RoboDK station: kr30 cnc 071219 julian curve.rdk

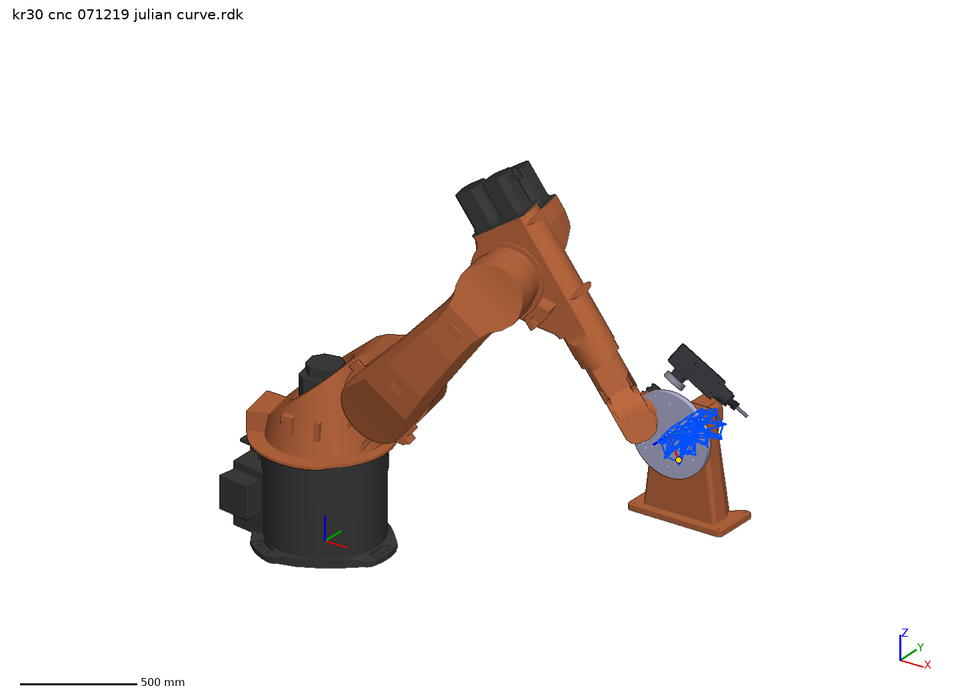
[picture v0: the station drawn from its stored meshes, robots at their saved joint values, targets as dots, program paths as lines]
Station kr30 cnc 071219 julian curve. Poses are relative to the parent item; angles as X-Y-Z fixed-axis rotations.
  - machining project Curve settings: C:/Temp/temp3/RhinoProject.stl | rotZ(0) | rotX(0)*rotY(0) | rotz(0) | onStart | onPathStart | onApproach | onPoint | onRetract | onFinish | onPathFinish | M_RunCode(%1)
  - frame KUKA KP1 MD250 Base at (0, 0, 0) mm
    - robot GIGASHEEN TURNTABLE OF DEATH: 1 axes, payload 250 kg
        modified DH rows (alpha deg, a mm, theta deg, d mm): 0, 0, 0, 0
        base shift (1587.22, 296.05, 828) mm, rotated rx 0 ry 90 rz -90 deg
        joint limits [-3600] to [3600]; home [0]; saved at [-332.14]
      - frame Reference Rhino at (0, 0, 0) mm
        - object RhinoPart at (0, -260, 100) mm
        - object Test Piece at (0, 0, 0) mm, geometry from Test Piece.stp
  - frame KUKA KR 30 HA Base at (0, 0, 0) mm
    - robot KUKA KR 30 HA: 6 axes, payload 30 kg, reach 2033 mm, repeatability 0.05 mm, weight 665 kg
        modified DH rows (alpha deg, a mm, theta deg, d mm): 0, 0, 0, 815; -90, 350, 0, 0; 0, 850, -90, 0; -90, 145, 0, 820; 90, 0, 0, 0; -90, 0, 180, 170
        joint limits [-185, -135, -120, -350, -119, -350] to [185, 35, 158, 350, 119, 350]; home [0, -90, 90, 0, 0, 0]; saved at [-11.373, -50.021, 107.833, -147.844, 108.332, -176.467]
      - tool 1/2" End Mill TCP, TCP at (337.71, -2.2, 160.57) mm, rotated rx 0 ry 90 rz 0 deg, size 415.8 x 102 x 153.6 mm
  - machining project RhinoPart Settings: rotZ(0) | rotX(90)*rotY(-155) | rotz(0)
  - program RhinoPart (1768 instructions, listed below)
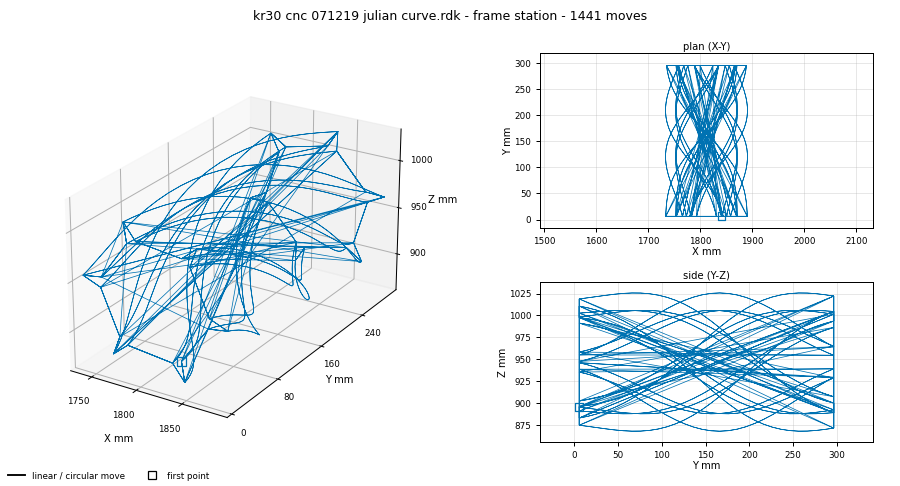
[picture p0: tool path of kr30 cnc 071219 julian curve.rdk in frame station, 1441 of 1441 moves have a stored position in this frame; points joined in program order, loops and branches not executed]

--- program RhinoPart (robot KUKA KR 30 HA) ---
  Set Ref.: Reference Rhino
  Set Tool: 1/2" End Mill TCP
  Show 1/2" End Mill TCP
  Set speed (1000.0 mm/s)
  MoveJ 1 to (58.93, 255.88, 290) mm, rotated rx -90 ry -25 rz 136 deg; joints [-2.265, -48.411, 103.049, -142.26, 108.636, -182.753, -175.998]
  MoveL 2 to (58.93, 255.88, 290) mm, rotated rx -90 ry -25 rz 136 deg; joints [-2.265, -48.411, 103.049, -142.26, 108.636, -182.753, -175.998]
  MoveL 3 to (58.93, 255.88, 290) mm, rotated rx -90 ry -25 rz 136 deg; joints [-2.265, -48.411, 103.049, -142.26, 108.636, -182.753, -175.998]
  Set speed (60.0 mm/s)
  MoveL 4 to (37.11, 300.24, 290) mm, rotated rx -90 ry -25 rz -172.69 deg; joints [-2.265, -48.205, 103.066, -142.213, 108.813, -182.608, -227.315]
  Set speed (1000.0 mm/s)
  MoveL 5 to (37.11, 300.24, 290) mm, rotated rx -90 ry -25 rz -172.69 deg; joints [-2.265, -48.205, 103.066, -142.213, 108.813, -182.608, -227.315]
  Set speed (1000.0 mm/s)
  MoveL 6 to (-37.11, 208.63, 290) mm, rotated rx -90 ry -25 rz 14.16 deg; joints [-2.265, -48.614, 103.03, -142.305, 108.461, -182.896, -54.156]
  MoveL 7 to (-37.11, 208.63, 290) mm, rotated rx -90 ry -25 rz 14.16 deg; joints [-2.265, -48.614, 103.03, -142.305, 108.461, -182.896, -54.156]
  Set speed (60.0 mm/s)
  MoveL 8 to (-58.93, 252.99, 290) mm, rotated rx -90 ry -25 rz -33.22 deg; joints [-2.265, -48.424, 103.048, -142.262, 108.625, -182.762, -6.784]
  Set speed (1000.0 mm/s)
  MoveL 9 to (-58.93, 252.99, 290) mm, rotated rx -90 ry -25 rz -33.22 deg; joints [-2.265, -48.424, 103.048, -142.262, 108.625, -182.762, -6.784]
  Set speed (1000.0 mm/s)
  MoveL 10 to (21.11, 199.39, 290) mm, rotated rx -90 ry -25 rz 69.21 deg; joints [-2.265, -48.652, 103.027, -142.314, 108.428, -182.923, -109.206]
  MoveL 11 to (21.11, 199.39, 290) mm, rotated rx -90 ry -25 rz 69.21 deg; joints [-2.265, -48.652, 103.027, -142.314, 108.428, -182.923, -109.206]
  Set speed (60.0 mm/s)
  MoveL 12 to (34.79, 183.72, 290) mm, rotated rx -90 ry -25 rz 74.51 deg; joints [-2.265, -49.571, 102.922, -142.517, 107.617, -183.579, -114.515]
  Set speed (1000.0 mm/s)
  MoveL 13 to (34.79, 183.72, 290) mm, rotated rx -90 ry -25 rz 74.51 deg; joints [-2.265, -49.571, 102.922, -142.517, 107.617, -183.579, -114.515]
  Set speed (1000.0 mm/s)
  MoveL 14 to (21.11, 199.39, 290) mm, rotated rx -90 ry -25 rz 69.21 deg; joints [-2.265, -48.652, 103.027, -142.314, 108.428, -182.923, -109.206]
  MoveL 15 to (21.11, 199.39, 290) mm, rotated rx -90 ry -25 rz 69.21 deg; joints [-2.265, -48.652, 103.027, -142.314, 108.428, -182.923, -109.206]
  Set speed (60.0 mm/s)
  MoveL 16 to (-28.22, 202.67, 290) mm, rotated rx -90 ry -25 rz 23.79 deg; joints [-2.265, -48.639, 103.028, -142.311, 108.44, -182.913, -63.793]
  Set speed (1000.0 mm/s)
  MoveL 17 to (-28.22, 202.67, 290) mm, rotated rx -90 ry -25 rz 23.79 deg; joints [-2.265, -48.639, 103.028, -142.311, 108.44, -182.913, -63.793]
  Set speed (1000.0 mm/s)
  MoveL 18 to (-43.85, 188.95, 290) mm, rotated rx -90 ry -25 rz 18.32 deg; joints [-2.265, -49.555, 102.924, -142.513, 107.631, -183.568, -58.321]
  MoveL 19 to (-43.85, 188.95, 290) mm, rotated rx -90 ry -25 rz 18.32 deg; joints [-2.265, -49.555, 102.924, -142.513, 107.631, -183.568, -58.321]
  Set speed (60.0 mm/s)
  MoveL 20 to (-28.22, 202.67, 290) mm, rotated rx -90 ry -25 rz 23.79 deg; joints [-2.265, -48.639, 103.028, -142.311, 108.44, -182.913, -63.793]
  Set speed (1000.0 mm/s)
  MoveL 21 to (-28.22, 202.67, 290) mm, rotated rx -90 ry -25 rz 23.79 deg; joints [-2.265, -48.639, 103.028, -142.311, 108.44, -182.913, -63.793]
  Set speed (1000.0 mm/s)
  MoveL 22 to (-43.85, 188.95, 290) mm, rotated rx -90 ry -25 rz 18.32 deg; joints [-2.265, -49.555, 102.924, -142.513, 107.631, -183.568, -58.321]
  MoveL 23 to (-43.85, 188.95, 290) mm, rotated rx -90 ry -25 rz 18.32 deg; joints [-2.265, -49.555, 102.924, -142.513, 107.631, -183.568, -58.321]
  Set speed (60.0 mm/s)
  MoveL 24 to (-37.11, 208.63, 290) mm, rotated rx -90 ry -25 rz 14.16 deg; joints [-2.265, -48.614, 103.03, -142.305, 108.461, -182.896, -54.156]
  Set speed (1000.0 mm/s)
  MoveL 25 to (-37.11, 208.63, 290) mm, rotated rx -90 ry -25 rz 14.16 deg; joints [-2.265, -48.614, 103.03, -142.305, 108.461, -182.896, -54.156]
  Set speed (1000.0 mm/s)
  MoveL 26 to (-78.63, 259.66, 290) mm, rotated rx -90 ry -25 rz -39.75 deg; joints [-2.265, -49.329, 102.952, -142.464, 107.833, -183.405, -0.245]
  MoveL 27 to (-78.63, 259.66, 290) mm, rotated rx -90 ry -25 rz -39.75 deg; joints [-2.265, -49.329, 102.952, -142.464, 107.833, -183.405, -0.245]
  Set speed (60.0 mm/s)
  MoveL 28 to (-58.93, 252.99, 290) mm, rotated rx -90 ry -25 rz -33.22 deg; joints [-2.265, -48.424, 103.048, -142.262, 108.625, -182.762, -6.784]
  Set speed (1000.0 mm/s)
  MoveL 29 to (-58.93, 252.99, 290) mm, rotated rx -90 ry -25 rz -33.22 deg; joints [-2.265, -48.424, 103.048, -142.262, 108.625, -182.762, -6.784]
  Set speed (1000.0 mm/s)
  MoveL 30 to (-78.63, 259.66, 290) mm, rotated rx -90 ry -25 rz -39.75 deg; joints [-2.265, -49.329, 102.952, -142.464, 107.833, -183.405, -0.245]
  MoveL 31 to (-78.63, 259.66, 290) mm, rotated rx -90 ry -25 rz -39.75 deg; joints [-2.265, -49.329, 102.952, -142.464, 107.833, -183.405, -0.245]
  Set speed (60.0 mm/s)
  MoveL 32 to (-58.22, 263.67, 290) mm, rotated rx -90 ry -25 rz -43.61 deg; joints [-2.265, -48.376, 103.052, -142.252, 108.666, -182.728, 3.606]
  Set speed (1000.0 mm/s)
  MoveL 33 to (-58.22, 263.67, 290) mm, rotated rx -90 ry -25 rz -43.61 deg; joints [-2.265, -48.376, 103.052, -142.252, 108.666, -182.728, 3.606]
  Set speed (1000.0 mm/s)
  MoveL 34 to (-30.72, 304.75, 290) mm, rotated rx -90 ry -25 rz -95.53 deg; joints [-2.265, -48.183, 103.068, -142.208, 108.831, -182.593, 55.533]
  MoveL 35 to (-30.72, 304.75, 290) mm, rotated rx -90 ry -25 rz -95.53 deg; joints [-2.265, -48.183, 103.068, -142.208, 108.831, -182.593, 55.533]
  Set speed (60.0 mm/s)
  MoveL 36 to (-58.22, 263.67, 290) mm, rotated rx -90 ry -25 rz -43.61 deg; joints [-2.265, -48.376, 103.052, -142.252, 108.666, -182.728, 3.606]
  Set speed (1000.0 mm/s)
  MoveL 37 to (-58.22, 263.67, 290) mm, rotated rx -90 ry -25 rz -43.61 deg; joints [-2.265, -48.376, 103.052, -142.252, 108.666, -182.728, 3.606]
  Set speed (1000.0 mm/s)
  MoveL 38 to (-30.72, 304.75, 290) mm, rotated rx -90 ry -25 rz -95.53 deg; joints [-2.265, -48.183, 103.068, -142.208, 108.831, -182.593, 55.533]
  MoveL 39 to (-30.72, 304.75, 290) mm, rotated rx -90 ry -25 rz -95.53 deg; joints [-2.265, -48.183, 103.068, -142.208, 108.831, -182.593, 55.533]
  Set speed (60.0 mm/s)
  MoveL 40 to (-34.79, 325.15, 290) mm, rotated rx -90 ry -25 rz -101.9 deg; joints [-2.265, -49.106, 102.979, -142.415, 108.03, -183.245, 61.899]
  Set speed (1000.0 mm/s)
  MoveL 41 to (-34.79, 325.15, 290) mm, rotated rx -90 ry -25 rz -101.9 deg; joints [-2.265, -49.106, 102.979, -142.415, 108.03, -183.245, 61.899]
  Set speed (1000.0 mm/s)
  MoveL 42 to (-21.11, 309.47, 290) mm, rotated rx -90 ry -25 rz -106.89 deg; joints [-2.265, -48.16, 103.069, -142.203, 108.851, -182.577, 66.89]
  MoveL 43 to (-21.11, 309.47, 290) mm, rotated rx -90 ry -25 rz -106.89 deg; joints [-2.265, -48.16, 103.069, -142.203, 108.851, -182.577, 66.89]
  Set speed (60.0 mm/s)
  MoveL 44 to (-34.79, 325.15, 290) mm, rotated rx -90 ry -25 rz -101.9 deg; joints [-2.265, -49.106, 102.979, -142.415, 108.03, -183.245, 61.899]
  Set speed (1000.0 mm/s)
  MoveL 45 to (-34.79, 325.15, 290) mm, rotated rx -90 ry -25 rz -101.9 deg; joints [-2.265, -49.106, 102.979, -142.415, 108.03, -183.245, 61.899]
  Set speed (1000.0 mm/s)
  MoveL 46 to (-21.11, 309.47, 290) mm, rotated rx -90 ry -25 rz -106.89 deg; joints [-2.265, -48.16, 103.069, -142.203, 108.851, -182.577, 66.89]
  MoveL 47 to (-21.11, 309.47, 290) mm, rotated rx -90 ry -25 rz -106.89 deg; joints [-2.265, -48.16, 103.069, -142.203, 108.851, -182.577, 66.89]
  Set speed (60.0 mm/s)
  MoveL 48 to (28.22, 306.19, 290) mm, rotated rx -90 ry -25 rz -161.42 deg; joints [-2.265, -48.176, 103.068, -142.207, 108.838, -182.588, 121.418]
  Set speed (1000.0 mm/s)
  MoveL 49 to (28.22, 306.19, 290) mm, rotated rx -90 ry -25 rz -161.42 deg; joints [-2.265, -48.176, 103.068, -142.207, 108.838, -182.588, 121.418]
  Set speed (1000.0 mm/s)
  MoveL 50 to (43.85, 319.91, 290) mm, rotated rx -90 ry -25 rz -166.2 deg; joints [-2.265, -49.125, 102.977, -142.419, 108.014, -183.258, 126.197]
  MoveL 51 to (43.85, 319.91, 290) mm, rotated rx -90 ry -25 rz -166.2 deg; joints [-2.265, -49.125, 102.977, -142.419, 108.014, -183.258, 126.197]
  Set speed (60.0 mm/s)
  MoveL 52 to (28.22, 306.19, 290) mm, rotated rx -90 ry -25 rz -161.42 deg; joints [-2.265, -48.176, 103.068, -142.207, 108.838, -182.588, 121.418]
  Set speed (1000.0 mm/s)
  MoveL 53 to (28.22, 306.19, 290) mm, rotated rx -90 ry -25 rz -161.42 deg; joints [-2.265, -48.176, 103.068, -142.207, 108.838, -182.588, 121.418]
  Set speed (1000.0 mm/s)
  MoveL 54 to (43.85, 319.91, 290) mm, rotated rx -90 ry -25 rz -166.2 deg; joints [-2.265, -49.125, 102.977, -142.419, 108.014, -183.258, 126.197]
  MoveL 55 to (43.85, 319.91, 290) mm, rotated rx -90 ry -25 rz -166.2 deg; joints [-2.265, -49.125, 102.977, -142.419, 108.014, -183.258, 126.197]
  Set speed (60.0 mm/s)
  MoveL 56 to (37.11, 300.24, 290) mm, rotated rx -90 ry -25 rz -172.69 deg; joints [-2.265, -48.205, 103.066, -142.213, 108.813, -182.608, 132.685]
  Set speed (1000.0 mm/s)
  MoveL 57 to (37.11, 300.24, 290) mm, rotated rx -90 ry -25 rz -172.69 deg; joints [-2.265, -48.205, 103.066, -142.213, 108.813, -182.608, 132.685]
  Set speed (1000.0 mm/s)
  MoveL 58 to (78.63, 249.2, 290) mm, rotated rx -90 ry -25 rz 132.18 deg; joints [-2.265, -49.364, 102.948, -142.471, 107.802, -183.43, 187.819]
  MoveL 59 to (78.63, 249.2, 290) mm, rotated rx -90 ry -25 rz 132.18 deg; joints [-2.265, -49.364, 102.948, -142.471, 107.802, -183.43, 187.819]
  Set speed (60.0 mm/s)
  MoveL 60 to (58.93, 255.88, 290) mm, rotated rx -90 ry -25 rz 136 deg; joints [-2.265, -48.411, 103.049, -142.26, 108.636, -182.753, 184.002]
  Set speed (1000.0 mm/s)
  MoveL 61 to (58.93, 255.88, 290) mm, rotated rx -90 ry -25 rz 136 deg; joints [-2.265, -48.411, 103.049, -142.26, 108.636, -182.753, 184.002]
  Set speed (1000.0 mm/s)
  MoveL 62 to (78.63, 249.2, 290) mm, rotated rx -90 ry -25 rz 132.18 deg; joints [-2.265, -49.364, 102.948, -142.471, 107.802, -183.43, 187.819]
  MoveL 63 to (78.63, 249.2, 290) mm, rotated rx -90 ry -25 rz 132.18 deg; joints [-2.265, -49.364, 102.948, -142.471, 107.802, -183.43, 187.819]
  Set speed (60.0 mm/s)
  MoveL 64 to (58.22, 245.2, 290) mm, rotated rx -90 ry -25 rz 125.73 deg; joints [-2.265, -48.458, 103.045, -142.27, 108.596, -182.786, 194.265]
  Set speed (1000.0 mm/s)
  MoveL 65 to (58.22, 245.2, 290) mm, rotated rx -90 ry -25 rz 125.73 deg; joints [-2.265, -48.458, 103.045, -142.27, 108.596, -182.786, 194.265]
  Set speed (1000.0 mm/s)
  MoveL 66 to (30.72, 204.12, 290) mm, rotated rx -90 ry -25 rz 78.8 deg; joints [-2.265, -48.633, 103.028, -142.309, 108.445, -182.909, 241.204]
  MoveL 67 to (30.72, 204.12, 290) mm, rotated rx -90 ry -25 rz 78.8 deg; joints [-2.265, -48.633, 103.028, -142.309, 108.445, -182.909, 241.204]
  Set speed (60.0 mm/s)
  MoveL 68 to (58.22, 245.2, 290) mm, rotated rx -90 ry -25 rz 125.73 deg; joints [-2.265, -48.458, 103.045, -142.27, 108.596, -182.786, 194.265]
  Set speed (1000.0 mm/s)
  MoveL 69 to (58.22, 245.2, 290) mm, rotated rx -90 ry -25 rz 125.73 deg; joints [-2.265, -48.458, 103.045, -142.27, 108.596, -182.786, 194.265]
  Set speed (1000.0 mm/s)
  MoveL 70 to (30.72, 204.12, 290) mm, rotated rx -90 ry -25 rz 78.8 deg; joints [-2.265, -48.633, 103.028, -142.309, 108.445, -182.909, 241.204]
  MoveL 71 to (30.72, 204.12, 290) mm, rotated rx -90 ry -25 rz 78.8 deg; joints [-2.265, -48.633, 103.028, -142.309, 108.445, -182.909, 241.204]
  Set speed (60.0 mm/s)
  MoveL 72 to (34.79, 183.72, 290) mm, rotated rx -90 ry -25 rz 74.51 deg; joints [-2.265, -49.571, 102.922, -142.517, 107.617, -183.579, 245.485]
  Set speed (1000.0 mm/s)
  MoveL 73 to (34.79, 183.72, 290) mm, rotated rx -90 ry -25 rz 74.51 deg; joints [-2.265, -49.571, 102.922, -142.517, 107.617, -183.579, 245.485]
  Set speed (1000.0 mm/s)
  MoveL 74 to (-37.62, 299.82, 0) mm, rotated rx -90 ry -25 rz -86.62 deg; joints [-13.282, -51.1, 108.722, -149.208, 107.637, -175.657, 406.623]
  MoveL 75 to (-37.62, 299.82, 0) mm, rotated rx -90 ry -25 rz -86.62 deg; joints [-13.282, -51.1, 108.722, -149.208, 107.637, -175.657, 406.623]
  Set speed (60.0 mm/s)
  MoveL 76 to (10.16, 312.5, 0) mm, rotated rx -90 ry -25 rz -140.95 deg; joints [-13.282, -51.034, 108.727, -149.196, 107.698, -175.619, 460.953]
  Set speed (1000.0 mm/s)
  MoveL 77 to (10.16, 312.5, 0) mm, rotated rx -90 ry -25 rz -140.95 deg; joints [-13.282, -51.034, 108.727, -149.196, 107.698, -175.619, 460.953]
  Set speed (1000.0 mm/s)
  MoveL 78 to (-37.62, 299.82, 0) mm, rotated rx -90 ry -25 rz -86.62 deg; joints [-13.282, -51.1, 108.722, -149.208, 107.637, -175.657, 406.623]
  MoveL 79 to (-37.62, 299.82, 0) mm, rotated rx -90 ry -25 rz -86.62 deg; joints [-13.282, -51.1, 108.722, -149.208, 107.637, -175.657, 406.623]
  Set speed (60.0 mm/s)
  MoveL 80 to (-55.59, 310.29, 0) mm, rotated rx -90 ry -25 rz -72.13 deg; joints [-13.325, -47.71, 107.988, -147.352, 118.871, -169.368, 402.13]
  Set speed (1000.0 mm/s)
  MoveL 81 to (-55.59, 310.29, 0) mm, rotated rx -90 ry -25 rz -72.13 deg; joints [-13.325, -47.71, 107.988, -147.352, 118.871, -169.368, 402.13]
  Set speed (1000.0 mm/s)
  MoveL 82 to (-45.21, 292.27, 0) mm, rotated rx -90 ry -25 rz -75.52 deg; joints [-13.282, -51.139, 108.719, -149.215, 107.602, -175.679, 395.516]
  MoveL 83 to (-45.21, 292.27, 0) mm, rotated rx -90 ry -25 rz -75.52 deg; joints [-13.282, -51.139, 108.719, -149.215, 107.602, -175.679, 395.516]
  Set speed (60.0 mm/s)
  MoveL 84 to (-55.59, 310.29, 0) mm, rotated rx -90 ry -25 rz -72.13 deg; joints [-13.325, -47.71, 107.988, -147.352, 118.871, -169.368, 402.13]
  Set speed (1000.0 mm/s)
  MoveL 85 to (-55.59, 310.29, 0) mm, rotated rx -90 ry -25 rz -72.13 deg; joints [-13.325, -47.71, 107.988, -147.352, 118.871, -169.368, 402.13]
  Set speed (1000.0 mm/s)
  MoveL 86 to (-45.21, 292.27, 0) mm, rotated rx -90 ry -25 rz -75.52 deg; joints [-13.282, -51.139, 108.719, -149.215, 107.602, -175.679, 395.516]
  MoveL 87 to (-45.21, 292.27, 0) mm, rotated rx -90 ry -25 rz -75.52 deg; joints [-13.282, -51.139, 108.719, -149.215, 107.602, -175.679, 395.516]
  Set speed (60.0 mm/s)
  MoveL 88 to (-58.12, 244.54, 0) mm, rotated rx -90 ry -25 rz -25.11 deg; joints [-13.282, -51.369, 108.701, -149.255, 107.387, -175.813, 345.106]
  Set speed (1000.0 mm/s)
  MoveL 89 to (-58.12, 244.54, 0) mm, rotated rx -90 ry -25 rz -25.11 deg; joints [-13.282, -51.369, 108.701, -149.255, 107.387, -175.813, 345.106]
  Set speed (1000.0 mm/s)
  MoveL 90 to (-76.17, 234.21, 0) mm, rotated rx -90 ry -25 rz -11.3 deg; joints [-13.325, -47.995, 107.992, -147.435, 118.635, -169.541, 341.297]
  MoveL 91 to (-76.17, 234.21, 0) mm, rotated rx -90 ry -25 rz -11.3 deg; joints [-13.325, -47.995, 107.992, -147.435, 118.635, -169.541, 341.297]
  Set speed (60.0 mm/s)
  MoveL 92 to (-58.12, 244.54, 0) mm, rotated rx -90 ry -25 rz -25.11 deg; joints [-13.282, -51.369, 108.701, -149.255, 107.387, -175.813, 345.106]
  Set speed (1000.0 mm/s)
  MoveL 93 to (-58.12, 244.54, 0) mm, rotated rx -90 ry -25 rz -25.11 deg; joints [-13.282, -51.369, 108.701, -149.255, 107.387, -175.813, 345.106]
  Set speed (1000.0 mm/s)
  MoveL 94 to (-76.17, 234.21, 0) mm, rotated rx -90 ry -25 rz -11.3 deg; joints [-13.325, -47.995, 107.992, -147.435, 118.635, -169.541, 341.297]
  MoveL 95 to (-76.17, 234.21, 0) mm, rotated rx -90 ry -25 rz -11.3 deg; joints [-13.325, -47.995, 107.992, -147.435, 118.635, -169.541, 341.297]
  Set speed (60.0 mm/s)
  MoveL 96 to (-55.37, 234.2, 0) mm, rotated rx -90 ry -25 rz -15.01 deg; joints [-13.282, -51.417, 108.696, -149.263, 107.343, -175.84, 335.014]
  Set speed (1000.0 mm/s)
  MoveL 97 to (-55.37, 234.2, 0) mm, rotated rx -90 ry -25 rz -15.01 deg; joints [-13.282, -51.417, 108.696, -149.263, 107.343, -175.84, 335.014]
  Set speed (1000.0 mm/s)
  MoveL 98 to (-20.49, 199.16, 0) mm, rotated rx -90 ry -25 rz 31.39 deg; joints [-13.282, -51.572, 108.683, -149.29, 107.197, -175.931, 288.615]
  MoveL 99 to (-20.49, 199.16, 0) mm, rotated rx -90 ry -25 rz 31.39 deg; joints [-13.282, -51.572, 108.683, -149.29, 107.197, -175.931, 288.615]
  Set speed (60.0 mm/s)
  MoveL 100 to (-55.37, 234.2, 0) mm, rotated rx -90 ry -25 rz -15.01 deg; joints [-13.282, -51.417, 108.696, -149.263, 107.343, -175.84, 335.014]
  Set speed (1000.0 mm/s)
  MoveL 101 to (-55.37, 234.2, 0) mm, rotated rx -90 ry -25 rz -15.01 deg; joints [-13.282, -51.417, 108.696, -149.263, 107.343, -175.84, 335.014]
  Set speed (1000.0 mm/s)
  MoveL 102 to (-20.49, 199.16, 0) mm, rotated rx -90 ry -25 rz 31.39 deg; joints [-13.282, -51.572, 108.683, -149.29, 107.197, -175.931, 288.615]
  MoveL 103 to (-20.49, 199.16, 0) mm, rotated rx -90 ry -25 rz 31.39 deg; joints [-13.282, -51.572, 108.683, -149.29, 107.197, -175.931, 288.615]
  Set speed (60.0 mm/s)
  MoveL 104 to (-20.57, 178.36, 0) mm, rotated rx -90 ry -25 rz 45.86 deg; joints [-13.325, -48.191, 107.994, -147.492, 118.47, -169.661, 284.144]
  Set speed (1000.0 mm/s)
  MoveL 105 to (-20.57, 178.36, 0) mm, rotated rx -90 ry -25 rz 45.86 deg; joints [-13.325, -48.191, 107.994, -147.492, 118.47, -169.661, 284.144]
  Set speed (1000.0 mm/s)
  MoveL 106 to (-10.16, 196.36, 0) mm, rotated rx -90 ry -25 rz 40.93 deg; joints [-13.282, -51.585, 108.681, -149.292, 107.186, -175.938, 279.071]
  MoveL 107 to (-10.16, 196.36, 0) mm, rotated rx -90 ry -25 rz 40.93 deg; joints [-13.282, -51.585, 108.681, -149.292, 107.186, -175.938, 279.071]
  Set speed (60.0 mm/s)
  MoveL 108 to (-20.57, 178.36, 0) mm, rotated rx -90 ry -25 rz 45.86 deg; joints [-13.325, -48.191, 107.994, -147.492, 118.47, -169.661, 284.144]
  Set speed (1000.0 mm/s)
  MoveL 109 to (-20.57, 178.36, 0) mm, rotated rx -90 ry -25 rz 45.86 deg; joints [-13.325, -48.191, 107.994, -147.492, 118.47, -169.661, 284.144]
  Set speed (1000.0 mm/s)
  MoveL 110 to (-10.16, 196.36, 0) mm, rotated rx -90 ry -25 rz 40.93 deg; joints [-13.282, -51.585, 108.681, -149.292, 107.186, -175.938, 279.071]
  MoveL 111 to (-10.16, 196.36, 0) mm, rotated rx -90 ry -25 rz 40.93 deg; joints [-13.282, -51.585, 108.681, -149.292, 107.186, -175.938, 279.071]
  Set speed (60.0 mm/s)
  MoveL 112 to (37.62, 209.05, 0) mm, rotated rx -90 ry -25 rz 86.44 deg; joints [-13.282, -51.529, 108.687, -149.283, 107.238, -175.906, 233.558]
  Set speed (1000.0 mm/s)
  MoveL 113 to (37.62, 209.05, 0) mm, rotated rx -90 ry -25 rz 86.44 deg; joints [-13.282, -51.529, 108.687, -149.283, 107.238, -175.906, 233.558]
  Set speed (1000.0 mm/s)
  MoveL 114 to (55.59, 198.58, 0) mm, rotated rx -90 ry -25 rz 102.15 deg; joints [-13.325, -48.121, 107.993, -147.471, 118.529, -169.618, 227.85]
  MoveL 115 to (55.59, 198.58, 0) mm, rotated rx -90 ry -25 rz 102.15 deg; joints [-13.325, -48.121, 107.993, -147.471, 118.529, -169.618, 227.85]
  Set speed (60.0 mm/s)
  MoveL 116 to (37.62, 209.05, 0) mm, rotated rx -90 ry -25 rz 86.44 deg; joints [-13.282, -51.529, 108.687, -149.283, 107.238, -175.906, 233.558]
  Set speed (1000.0 mm/s)
  MoveL 117 to (37.62, 209.05, 0) mm, rotated rx -90 ry -25 rz 86.44 deg; joints [-13.282, -51.529, 108.687, -149.283, 107.238, -175.906, 233.558]
  Set speed (1000.0 mm/s)
  MoveL 118 to (55.59, 198.58, 0) mm, rotated rx -90 ry -25 rz 102.15 deg; joints [-13.325, -48.121, 107.993, -147.471, 118.529, -169.618, 227.85]
  MoveL 119 to (55.59, 198.58, 0) mm, rotated rx -90 ry -25 rz 102.15 deg; joints [-13.325, -48.121, 107.993, -147.471, 118.529, -169.618, 227.85]
  Set speed (60.0 mm/s)
  MoveL 120 to (45.21, 216.6, 0) mm, rotated rx -90 ry -25 rz 96.17 deg; joints [-13.282, -51.496, 108.69, -149.277, 107.269, -175.887, 223.831]
  Set speed (1000.0 mm/s)
  MoveL 121 to (45.21, 216.6, 0) mm, rotated rx -90 ry -25 rz 96.17 deg; joints [-13.282, -51.496, 108.69, -149.277, 107.269, -175.887, 223.831]
  Set speed (1000.0 mm/s)
  MoveL 122 to (58.12, 264.32, 0) mm, rotated rx -90 ry -25 rz 144.25 deg; joints [-13.282, -51.276, 108.708, -149.239, 107.474, -175.759, 175.746]
  MoveL 123 to (58.12, 264.32, 0) mm, rotated rx -90 ry -25 rz 144.25 deg; joints [-13.282, -51.276, 108.708, -149.239, 107.474, -175.759, 175.746]
  Set speed (60.0 mm/s)
  MoveL 124 to (45.21, 216.6, 0) mm, rotated rx -90 ry -25 rz 96.17 deg; joints [-13.282, -51.496, 108.69, -149.277, 107.269, -175.887, 223.831]
  Set speed (1000.0 mm/s)
  MoveL 125 to (45.21, 216.6, 0) mm, rotated rx -90 ry -25 rz 96.17 deg; joints [-13.282, -51.496, 108.69, -149.277, 107.269, -175.887, 223.831]
  Set speed (1000.0 mm/s)
  MoveL 126 to (58.12, 264.32, 0) mm, rotated rx -90 ry -25 rz 144.25 deg; joints [-13.282, -51.276, 108.708, -149.239, 107.474, -175.759, 175.746]
  MoveL 127 to (58.12, 264.32, 0) mm, rotated rx -90 ry -25 rz 144.25 deg; joints [-13.282, -51.276, 108.708, -149.239, 107.474, -175.759, 175.746]
  Set speed (60.0 mm/s)
  MoveL 128 to (76.17, 274.65, 0) mm, rotated rx -90 ry -25 rz 160.89 deg; joints [-13.325, -47.846, 107.991, -147.391, 118.758, -169.451, 169.111]
  Set speed (1000.0 mm/s)
  MoveL 129 to (76.17, 274.65, 0) mm, rotated rx -90 ry -25 rz 160.89 deg; joints [-13.325, -47.846, 107.991, -147.391, 118.758, -169.451, 169.111]
  Set speed (1000.0 mm/s)
  MoveL 130 to (55.37, 274.67, 0) mm, rotated rx -90 ry -25 rz 154.84 deg; joints [-13.282, -51.226, 108.712, -149.23, 107.521, -175.73, 165.162]
  MoveL 131 to (55.37, 274.67, 0) mm, rotated rx -90 ry -25 rz 154.84 deg; joints [-13.282, -51.226, 108.712, -149.23, 107.521, -175.73, 165.162]
  Set speed (60.0 mm/s)
  MoveL 132 to (76.17, 274.65, 0) mm, rotated rx -90 ry -25 rz 160.89 deg; joints [-13.325, -47.846, 107.991, -147.391, 118.758, -169.451, 169.111]
  Set speed (1000.0 mm/s)
  MoveL 133 to (76.17, 274.65, 0) mm, rotated rx -90 ry -25 rz 160.89 deg; joints [-13.325, -47.846, 107.991, -147.391, 118.758, -169.451, 169.111]
  Set speed (1000.0 mm/s)
  MoveL 134 to (55.37, 274.67, 0) mm, rotated rx -90 ry -25 rz 154.84 deg; joints [-13.282, -51.226, 108.712, -149.23, 107.521, -175.73, 165.162]
  MoveL 135 to (55.37, 274.67, 0) mm, rotated rx -90 ry -25 rz 154.84 deg; joints [-13.282, -51.226, 108.712, -149.23, 107.521, -175.73, 165.162]
  Set speed (60.0 mm/s)
  MoveL 136 to (20.49, 309.71, 0) mm, rotated rx -90 ry -25 rz -152.4 deg; joints [-13.282, -51.049, 108.726, -149.199, 107.684, -175.627, 112.405]
  Set speed (1000.0 mm/s)
  MoveL 137 to (20.49, 309.71, 0) mm, rotated rx -90 ry -25 rz -152.4 deg; joints [-13.282, -51.049, 108.726, -149.199, 107.684, -175.627, 112.405]
  Set speed (1000.0 mm/s)
  MoveL 138 to (20.57, 330.51, 0) mm, rotated rx -90 ry -25 rz -136.27 deg; joints [-13.325, -47.631, 107.987, -147.328, 118.937, -169.32, 106.267]
  MoveL 139 to (20.57, 330.51, 0) mm, rotated rx -90 ry -25 rz -136.27 deg; joints [-13.325, -47.631, 107.987, -147.328, 118.937, -169.32, 106.267]
  Set speed (60.0 mm/s)
  MoveL 140 to (20.49, 309.71, 0) mm, rotated rx -90 ry -25 rz -152.4 deg; joints [-13.282, -51.049, 108.726, -149.199, 107.684, -175.627, 112.405]
  Set speed (1000.0 mm/s)
  MoveL 141 to (20.49, 309.71, 0) mm, rotated rx -90 ry -25 rz -152.4 deg; joints [-13.282, -51.049, 108.726, -149.199, 107.684, -175.627, 112.405]
  Set speed (1000.0 mm/s)
  MoveL 142 to (20.57, 330.51, 0) mm, rotated rx -90 ry -25 rz -136.27 deg; joints [-13.325, -47.631, 107.987, -147.328, 118.937, -169.32, 106.267]
  MoveL 143 to (20.57, 330.51, 0) mm, rotated rx -90 ry -25 rz -136.27 deg; joints [-13.325, -47.631, 107.987, -147.328, 118.937, -169.32, 106.267]
  Set speed (60.0 mm/s)
  MoveL 144 to (10.16, 312.5, 0) mm, rotated rx -90 ry -25 rz -140.95 deg; joints [-13.282, -51.034, 108.727, -149.196, 107.698, -175.619, 100.953]
  Set speed (1000.0 mm/s)
  MoveL 145 to (10.16, 312.5, 0) mm, rotated rx -90 ry -25 rz -140.95 deg; joints [-13.282, -51.034, 108.727, -149.196, 107.698, -175.619, 100.953]
  Set speed (1000.0 mm/s)
  MoveL 146 to (-37.62, 299.82, 0) mm, rotated rx -90 ry -25 rz -86.62 deg; joints [-13.282, -51.1, 108.722, -149.208, 107.637, -175.657, 46.623]
  MoveL 147 to (-37.62, 299.82, 0) mm, rotated rx -90 ry -25 rz -86.62 deg; joints [-13.282, -51.1, 108.722, -149.208, 107.637, -175.657, 46.623]
  Set speed (60.0 mm/s)
  MoveL 148 to (-40.85, 296.93, 10) mm, rotated rx -90 ry -25 rz -82.11 deg; joints [-12.889, -51.06, 108.613, -148.945, 107.687, -175.884, 42.114]
  MoveL 149 to (-44.15, 293.5, 20) mm, rotated rx -90 ry -25 rz -77.19 deg; joints [-12.496, -51.018, 108.497, -148.683, 107.732, -176.113, 37.19]
  MoveL 150 to (-47.39, 289.5, 30) mm, rotated rx -90 ry -25 rz -71.9 deg; joints [-12.104, -50.977, 108.376, -148.424, 107.774, -176.346, 31.9]
  MoveL 151 to (-50.45, 284.92, 40) mm, rotated rx -90 ry -25 rz -66.29 deg; joints [-11.713, -50.934, 108.247, -148.167, 107.811, -176.583, 26.29]
  MoveL 152 to (-53.21, 279.8, 50) mm, rotated rx -90 ry -25 rz -60.41 deg; joints [-11.323, -50.891, 108.112, -147.911, 107.845, -176.822, 20.409]
  MoveL 153 to (-55.55, 274.16, 60) mm, rotated rx -90 ry -25 rz -54.3 deg; joints [-10.933, -50.847, 107.971, -147.658, 107.876, -177.064, 14.303]
  MoveL 154 to (-57.35, 268.08, 70) mm, rotated rx -90 ry -25 rz -48.01 deg; joints [-10.544, -50.802, 107.823, -147.407, 107.903, -177.309, 8.015]
  MoveL 155 to (-58.51, 261.62, 80) mm, rotated rx -90 ry -25 rz -41.59 deg; joints [-10.156, -50.755, 107.669, -147.158, 107.927, -177.557, 1.589]
  MoveL 156 to (-58.95, 254.91, 90) mm, rotated rx -90 ry -25 rz -35.06 deg; joints [-9.769, -50.705, 107.509, -146.911, 107.949, -177.807, -4.936]
  MoveL 157 to (-58.6, 248.05, 100) mm, rotated rx -90 ry -25 rz -28.48 deg; joints [-9.383, -50.653, 107.343, -146.666, 107.97, -178.059, -11.521]
  MoveL 158 to (-57.44, 241.19, 110) mm, rotated rx -90 ry -25 rz -21.87 deg; joints [-8.998, -50.597, 107.17, -146.422, 107.99, -178.312, -18.132]
  MoveL 159 to (-55.46, 234.45, 120) mm, rotated rx -90 ry -25 rz -15.26 deg; joints [-8.614, -50.536, 106.991, -146.181, 108.009, -178.566, -24.736]
  MoveL 160 to (-52.68, 227.97, 130) mm, rotated rx -90 ry -25 rz -8.7 deg; joints [-8.231, -50.471, 106.806, -145.941, 108.027, -178.822, -31.302]
  MoveL 161 to (-49.15, 221.88, 140) mm, rotated rx -90 ry -25 rz -2.2 deg; joints [-7.849, -50.401, 106.615, -145.702, 108.047, -179.078, -37.801]
  MoveL 162 to (-44.94, 216.28, 150) mm, rotated rx -90 ry -25 rz 4.21 deg; joints [-7.468, -50.325, 106.418, -145.465, 108.067, -179.334, -44.207]
  MoveL 163 to (-40.17, 211.29, 160) mm, rotated rx -90 ry -25 rz 10.49 deg; joints [-7.088, -50.242, 106.215, -145.229, 108.088, -179.59, -50.492]
  MoveL 164 to (-34.94, 206.95, 170) mm, rotated rx -90 ry -25 rz 16.63 deg; joints [-6.709, -50.154, 106.005, -144.995, 108.11, -179.845, -56.632]
  MoveL 165 to (-29.38, 203.32, 180) mm, rotated rx -90 ry -25 rz 22.6 deg; joints [-6.332, -50.059, 105.79, -144.763, 108.134, -180.101, -62.601]
  MoveL 166 to (-23.62, 200.42, 190) mm, rotated rx -90 ry -25 rz 28.37 deg; joints [-5.956, -49.958, 105.569, -144.531, 108.159, -180.356, -68.373]
  MoveL 167 to (-17.8, 198.23, 200) mm, rotated rx -90 ry -25 rz 33.92 deg; joints [-5.581, -49.851, 105.343, -144.302, 108.185, -180.611, -73.923]
  MoveL 168 to (-12.04, 196.73, 210) mm, rotated rx -90 ry -25 rz 39.22 deg; joints [-5.207, -49.737, 105.11, -144.073, 108.213, -180.865, -79.224]
  MoveL 169 to (-6.46, 195.84, 220) mm, rotated rx -90 ry -25 rz 44.25 deg; joints [-4.834, -49.618, 104.871, -143.847, 108.241, -181.12, -84.249]
  MoveL 170 to (-1.16, 195.49, 230) mm, rotated rx -90 ry -25 rz 48.97 deg; joints [-4.463, -49.493, 104.626, -143.622, 108.269, -181.374, -88.971]
  MoveL 171 to (3.78, 195.6, 240) mm, rotated rx -90 ry -25 rz 53.36 deg; joints [-4.093, -49.363, 104.375, -143.398, 108.298, -181.63, -93.359]
  MoveL 172 to (8.28, 196.07, 250) mm, rotated rx -90 ry -25 rz 57.38 deg; joints [-3.725, -49.228, 104.118, -143.177, 108.326, -181.885, -97.383]
  MoveL 173 to (12.3, 196.78, 260) mm, rotated rx -90 ry -25 rz 61.01 deg; joints [-3.358, -49.09, 103.854, -142.958, 108.354, -182.142, -101.013]
  MoveL 174 to (15.8, 197.64, 270) mm, rotated rx -90 ry -25 rz 64.21 deg; joints [-2.992, -48.947, 103.585, -142.741, 108.38, -182.401, -104.215]
  MoveL 175 to (18.74, 198.54, 280) mm, rotated rx -90 ry -25 rz 66.96 deg; joints [-2.628, -48.801, 103.309, -142.526, 108.405, -182.661, -106.957]
  MoveL 176 to (21.11, 199.39, 290) mm, rotated rx -90 ry -25 rz 69.21 deg; joints [-2.265, -48.652, 103.027, -142.314, 108.428, -182.923, -109.206]
  Set speed (1000.0 mm/s)
  MoveL 177 to (21.11, 199.39, 290) mm, rotated rx -90 ry -25 rz 69.21 deg; joints [-2.265, -48.652, 103.027, -142.314, 108.428, -182.923, -109.206]
  Set speed (1000.0 mm/s)
  MoveL 178 to (10.16, 312.5, 0) mm, rotated rx -90 ry -25 rz -140.95 deg; joints [-13.282, -51.034, 108.727, -149.196, 107.698, -175.619, -259.047]
  MoveL 179 to (10.16, 312.5, 0) mm, rotated rx -90 ry -25 rz -140.95 deg; joints [-13.282, -51.034, 108.727, -149.196, 107.698, -175.619, -259.047]
  Set speed (60.0 mm/s)
  MoveL 180 to (-37.62, 299.82, 0) mm, rotated rx -90 ry -25 rz -86.62 deg; joints [-13.282, -51.1, 108.722, -149.208, 107.637, -175.657, -313.377]
  Set speed (1000.0 mm/s)
  MoveL 181 to (-37.62, 299.82, 0) mm, rotated rx -90 ry -25 rz -86.62 deg; joints [-13.282, -51.1, 108.722, -149.208, 107.637, -175.657, -313.377]
  Set speed (1000.0 mm/s)
  MoveL 182 to (-28.22, 202.67, 290) mm, rotated rx -90 ry -25 rz 23.79 deg; joints [-2.265, -48.639, 103.028, -142.311, 108.44, -182.913, -423.793]
  MoveL 183 to (-28.22, 202.67, 290) mm, rotated rx -90 ry -25 rz 23.79 deg; joints [-2.265, -48.639, 103.028, -142.311, 108.44, -182.913, -423.793]
  Set speed (60.0 mm/s)
  MoveL 184 to (21.11, 199.39, 290) mm, rotated rx -90 ry -25 rz 69.21 deg; joints [-2.265, -48.652, 103.027, -142.314, 108.428, -182.923, -469.206]
  Set speed (1000.0 mm/s)
  MoveL 185 to (21.11, 199.39, 290) mm, rotated rx -90 ry -25 rz 69.21 deg; joints [-2.265, -48.652, 103.027, -142.314, 108.428, -182.923, -469.206]
  Set speed (1000.0 mm/s)
  MoveL 186 to (-28.22, 202.67, 290) mm, rotated rx -90 ry -25 rz 23.79 deg; joints [-2.265, -48.639, 103.028, -142.311, 108.44, -182.913, -423.793]
  MoveL 187 to (-28.22, 202.67, 290) mm, rotated rx -90 ry -25 rz 23.79 deg; joints [-2.265, -48.639, 103.028, -142.311, 108.44, -182.913, -423.793]
  Set speed (60.0 mm/s)
  MoveL 188 to (-30.4, 203.93, 280) mm, rotated rx -90 ry -25 rz 21.53 deg; joints [-2.628, -48.779, 103.311, -142.521, 108.424, -182.645, -421.533]
  MoveL 189 to (-33, 205.58, 270) mm, rotated rx -90 ry -25 rz 18.77 deg; joints [-2.992, -48.914, 103.588, -142.734, 108.409, -182.378, -418.768]
  MoveL 190 to (-35.92, 207.69, 260) mm, rotated rx -90 ry -25 rz 15.53 deg; joints [-3.358, -49.044, 103.858, -142.948, 108.393, -182.111, -415.528]
  MoveL 191 to (-39.07, 210.28, 250) mm, rotated rx -90 ry -25 rz 11.84 deg; joints [-3.725, -49.169, 104.123, -143.164, 108.378, -181.845, -411.841]
  MoveL 192 to (-42.34, 213.41, 240) mm, rotated rx -90 ry -25 rz 7.73 deg; joints [-4.093, -49.289, 104.382, -143.382, 108.363, -181.578, -407.735]
  MoveL 193 to (-45.62, 217.1, 230) mm, rotated rx -90 ry -25 rz 3.24 deg; joints [-4.463, -49.402, 104.634, -143.602, 108.349, -181.312, -403.236]
  MoveL 194 to (-48.8, 221.36, 220) mm, rotated rx -90 ry -25 rz -1.63 deg; joints [-4.834, -49.51, 104.881, -143.824, 108.336, -181.046, -398.371]
  MoveL 195 to (-51.74, 226.19, 210) mm, rotated rx -90 ry -25 rz -6.84 deg; joints [-5.207, -49.612, 105.121, -144.047, 108.324, -180.781, -393.164]
  MoveL 196 to (-54.33, 231.55, 200) mm, rotated rx -90 ry -25 rz -12.36 deg; joints [-5.581, -49.708, 105.356, -144.272, 108.312, -180.515, -387.64]
  MoveL 197 to (-56.44, 237.4, 190) mm, rotated rx -90 ry -25 rz -18.18 deg; joints [-5.956, -49.798, 105.584, -144.498, 108.301, -180.249, -381.825]
  MoveL 198 to (-57.96, 243.66, 180) mm, rotated rx -90 ry -25 rz -24.26 deg; joints [-6.332, -49.883, 105.806, -144.726, 108.291, -179.984, -375.742]
  MoveL 199 to (-58.8, 250.25, 170) mm, rotated rx -90 ry -25 rz -30.58 deg; joints [-6.709, -49.963, 106.022, -144.956, 108.28, -179.72, -369.418]
  MoveL 200 to (-58.89, 257.04, 160) mm, rotated rx -90 ry -25 rz -37.12 deg; joints [-7.088, -50.039, 106.232, -145.188, 108.27, -179.457, -362.877]
  MoveL 201 to (-58.18, 263.92, 150) mm, rotated rx -90 ry -25 rz -43.85 deg; joints [-7.468, -50.11, 106.436, -145.422, 108.259, -179.194, -356.149]
  MoveL 202 to (-56.65, 270.74, 140) mm, rotated rx -90 ry -25 rz -50.74 deg; joints [-7.849, -50.178, 106.634, -145.657, 108.246, -178.934, -349.263]
  MoveL 203 to (-54.3, 277.38, 130) mm, rotated rx -90 ry -25 rz -57.75 deg; joints [-8.231, -50.243, 106.825, -145.895, 108.232, -178.676, -342.251]
  MoveL 204 to (-51.17, 283.7, 120) mm, rotated rx -90 ry -25 rz -64.85 deg; joints [-8.614, -50.306, 107.01, -146.135, 108.216, -178.42, -335.149]
  MoveL 205 to (-47.33, 289.58, 110) mm, rotated rx -90 ry -25 rz -72.01 deg; joints [-8.998, -50.368, 107.189, -146.378, 108.196, -178.168, -327.994]
  MoveL 206 to (-42.85, 294.92, 100) mm, rotated rx -90 ry -25 rz -79.17 deg; joints [-9.383, -50.428, 107.361, -146.622, 108.173, -177.918, -320.828]
  MoveL 207 to (-37.86, 299.62, 90) mm, rotated rx -90 ry -25 rz -86.3 deg; joints [-9.769, -50.489, 107.527, -146.869, 108.146, -177.672, -313.695]
  MoveL 208 to (-32.46, 303.64, 80) mm, rotated rx -90 ry -25 rz -93.36 deg; joints [-10.156, -50.549, 107.686, -147.119, 108.114, -177.43, -306.643]
  MoveL 209 to (-26.8, 306.94, 70) mm, rotated rx -90 ry -25 rz -100.28 deg; joints [-10.544, -50.61, 107.839, -147.371, 108.078, -177.191, -299.72]
  MoveL 210 to (-21, 309.52, 60) mm, rotated rx -90 ry -25 rz -107.02 deg; joints [-10.933, -50.671, 107.985, -147.625, 108.037, -176.957, -292.977]
  MoveL 211 to (-15.19, 311.39, 50) mm, rotated rx -90 ry -25 rz -113.54 deg; joints [-11.323, -50.732, 108.125, -147.882, 107.991, -176.726, -286.464]
  MoveL 212 to (-9.5, 312.61, 40) mm, rotated rx -90 ry -25 rz -119.77 deg; joints [-11.713, -50.794, 108.258, -148.141, 107.94, -176.499, -280.231]
  MoveL 213 to (-4.03, 313.25, 30) mm, rotated rx -90 ry -25 rz -125.67 deg; joints [-12.104, -50.855, 108.385, -148.402, 107.885, -176.275, -274.327]
  MoveL 214 to (1.12, 313.37, 20) mm, rotated rx -90 ry -25 rz -131.2 deg; joints [-12.496, -50.916, 108.505, -148.665, 107.826, -176.053, -268.799]
  MoveL 215 to (5.87, 313.09, 10) mm, rotated rx -90 ry -25 rz -136.31 deg; joints [-12.889, -50.976, 108.619, -148.93, 107.764, -175.835, -263.692]
  MoveL 216 to (10.16, 312.5, 0) mm, rotated rx -90 ry -25 rz -140.95 deg; joints [-13.282, -51.034, 108.727, -149.196, 107.698, -175.619, -259.047]
  Set speed (1000.0 mm/s)
  MoveL 217 to (10.16, 312.5, 0) mm, rotated rx -90 ry -25 rz -140.95 deg; joints [-13.282, -51.034, 108.727, -149.196, 107.698, -175.619, -259.047]
  Set speed (1000.0 mm/s)
  MoveL 218 to (-37.62, 299.82, 0) mm, rotated rx -90 ry -25 rz -86.62 deg; joints [-13.282, -51.1, 108.722, -149.208, 107.637, -175.657, -313.377]
  MoveL 219 to (-37.62, 299.82, 0) mm, rotated rx -90 ry -25 rz -86.62 deg; joints [-13.282, -51.1, 108.722, -149.208, 107.637, -175.657, -313.377]
  Set speed (60.0 mm/s)
  MoveL 220 to (-40.85, 296.93, 10) mm, rotated rx -90 ry -25 rz -82.11 deg; joints [-12.889, -51.06, 108.613, -148.945, 107.687, -175.884, -317.886]
  MoveL 221 to (-44.15, 293.5, 20) mm, rotated rx -90 ry -25 rz -77.19 deg; joints [-12.496, -51.018, 108.497, -148.683, 107.732, -176.113, -322.81]
  MoveL 222 to (-47.39, 289.5, 30) mm, rotated rx -90 ry -25 rz -71.9 deg; joints [-12.104, -50.977, 108.376, -148.424, 107.774, -176.346, -328.1]
  MoveL 223 to (-50.45, 284.92, 40) mm, rotated rx -90 ry -25 rz -66.29 deg; joints [-11.713, -50.934, 108.247, -148.167, 107.811, -176.583, -333.71]
  MoveL 224 to (-53.21, 279.8, 50) mm, rotated rx -90 ry -25 rz -60.41 deg; joints [-11.323, -50.891, 108.112, -147.911, 107.845, -176.822, -339.591]
  MoveL 225 to (-55.55, 274.16, 60) mm, rotated rx -90 ry -25 rz -54.3 deg; joints [-10.933, -50.847, 107.971, -147.658, 107.876, -177.064, -345.697]
  MoveL 226 to (-57.35, 268.08, 70) mm, rotated rx -90 ry -25 rz -48.01 deg; joints [-10.544, -50.802, 107.823, -147.407, 107.903, -177.309, -351.985]
  MoveL 227 to (-58.51, 261.62, 80) mm, rotated rx -90 ry -25 rz -41.59 deg; joints [-10.156, -50.755, 107.669, -147.158, 107.927, -177.557, -358.411]
  MoveL 228 to (-58.95, 254.91, 90) mm, rotated rx -90 ry -25 rz -35.06 deg; joints [-9.769, -50.705, 107.509, -146.911, 107.949, -177.807, -364.936]
  MoveL 229 to (-58.6, 248.05, 100) mm, rotated rx -90 ry -25 rz -28.48 deg; joints [-9.383, -50.653, 107.343, -146.666, 107.97, -178.059, -371.521]
  MoveL 230 to (-57.44, 241.19, 110) mm, rotated rx -90 ry -25 rz -21.87 deg; joints [-8.998, -50.597, 107.17, -146.422, 107.99, -178.312, -378.132]
  MoveL 231 to (-55.46, 234.45, 120) mm, rotated rx -90 ry -25 rz -15.26 deg; joints [-8.614, -50.536, 106.991, -146.181, 108.009, -178.566, -384.736]
  MoveL 232 to (-52.68, 227.97, 130) mm, rotated rx -90 ry -25 rz -8.7 deg; joints [-8.231, -50.471, 106.806, -145.941, 108.027, -178.822, -391.302]
  MoveL 233 to (-49.15, 221.88, 140) mm, rotated rx -90 ry -25 rz -2.2 deg; joints [-7.849, -50.401, 106.615, -145.702, 108.047, -179.078, -397.801]
  MoveL 234 to (-44.94, 216.28, 150) mm, rotated rx -90 ry -25 rz 4.21 deg; joints [-7.468, -50.325, 106.418, -145.465, 108.067, -179.334, -404.207]
  MoveL 235 to (-40.17, 211.29, 160) mm, rotated rx -90 ry -25 rz 10.49 deg; joints [-7.088, -50.242, 106.215, -145.229, 108.088, -179.59, -410.492]
  MoveL 236 to (-34.94, 206.95, 170) mm, rotated rx -90 ry -25 rz 16.63 deg; joints [-6.709, -50.154, 106.005, -144.995, 108.11, -179.845, -416.632]
  MoveL 237 to (-29.38, 203.32, 180) mm, rotated rx -90 ry -25 rz 22.6 deg; joints [-6.332, -50.059, 105.79, -144.763, 108.134, -180.101, -422.601]
  MoveL 238 to (-23.62, 200.42, 190) mm, rotated rx -90 ry -25 rz 28.37 deg; joints [-5.956, -49.958, 105.569, -144.531, 108.159, -180.356, -428.373]
  MoveL 239 to (-17.8, 198.23, 200) mm, rotated rx -90 ry -25 rz 33.92 deg; joints [-5.581, -49.851, 105.343, -144.302, 108.185, -180.611, -433.923]
  MoveL 240 to (-12.04, 196.73, 210) mm, rotated rx -90 ry -25 rz 39.22 deg; joints [-5.207, -49.737, 105.11, -144.073, 108.213, -180.865, -439.224]
  MoveL 241 to (-6.46, 195.84, 220) mm, rotated rx -90 ry -25 rz 44.25 deg; joints [-4.834, -49.618, 104.871, -143.847, 108.241, -181.12, -444.249]
  MoveL 242 to (-1.16, 195.49, 230) mm, rotated rx -90 ry -25 rz 48.97 deg; joints [-4.463, -49.493, 104.626, -143.622, 108.269, -181.374, -448.971]
  MoveL 243 to (3.78, 195.6, 240) mm, rotated rx -90 ry -25 rz 53.36 deg; joints [-4.093, -49.363, 104.375, -143.398, 108.298, -181.63, -453.359]
  MoveL 244 to (8.28, 196.07, 250) mm, rotated rx -90 ry -25 rz 57.38 deg; joints [-3.725, -49.228, 104.118, -143.177, 108.326, -181.885, -457.383]
  MoveL 245 to (12.3, 196.78, 260) mm, rotated rx -90 ry -25 rz 61.01 deg; joints [-3.358, -49.09, 103.854, -142.958, 108.354, -182.142, -461.013]
  MoveL 246 to (15.8, 197.64, 270) mm, rotated rx -90 ry -25 rz 64.21 deg; joints [-2.992, -48.947, 103.585, -142.741, 108.38, -182.401, -464.215]
  MoveL 247 to (18.74, 198.54, 280) mm, rotated rx -90 ry -25 rz 66.96 deg; joints [-2.628, -48.801, 103.309, -142.526, 108.405, -182.661, -466.957]
  MoveL 248 to (21.11, 199.39, 290) mm, rotated rx -90 ry -25 rz 69.21 deg; joints [-2.265, -48.652, 103.027, -142.314, 108.428, -182.923, -469.206]
  Set speed (1000.0 mm/s)
  MoveL 249 to (21.11, 199.39, 290) mm, rotated rx -90 ry -25 rz 69.21 deg; joints [-2.265, -48.652, 103.027, -142.314, 108.428, -182.923, -469.206]
  Set speed (1000.0 mm/s)
  MoveL 250 to (34.79, 183.72, 290) mm, rotated rx -90 ry -25 rz 74.51 deg; joints [-2.265, -49.571, 102.922, -142.517, 107.617, -183.579, -474.515]
  MoveL 251 to (34.79, 183.72, 290) mm, rotated rx -90 ry -25 rz 74.51 deg; joints [-2.265, -49.571, 102.922, -142.517, 107.617, -183.579, -474.515]
  Set speed (60.0 mm/s)
  MoveL 252 to (21.11, 199.39, 290) mm, rotated rx -90 ry -25 rz 69.21 deg; joints [-2.265, -48.652, 103.027, -142.314, 108.428, -182.923, -469.206]
  Set speed (1000.0 mm/s)
  MoveL 253 to (21.11, 199.39, 290) mm, rotated rx -90 ry -25 rz 69.21 deg; joints [-2.265, -48.652, 103.027, -142.314, 108.428, -182.923, -469.206]
  Set speed (1000.0 mm/s)
  MoveL 254 to (-55.59, 310.29, 0) mm, rotated rx -90 ry -25 rz -72.13 deg; joints [-13.325, -47.71, 107.988, -147.352, 118.871, -169.368, -317.87]
  MoveL 255 to (-55.59, 310.29, 0) mm, rotated rx -90 ry -25 rz -72.13 deg; joints [-13.325, -47.71, 107.988, -147.352, 118.871, -169.368, -317.87]
  Set speed (60.0 mm/s)
  MoveL 256 to (-37.62, 299.82, 0) mm, rotated rx -90 ry -25 rz -86.62 deg; joints [-13.282, -51.1, 108.722, -149.208, 107.637, -175.657, -313.377]
  Set speed (1000.0 mm/s)
  MoveL 257 to (-37.62, 299.82, 0) mm, rotated rx -90 ry -25 rz -86.62 deg; joints [-13.282, -51.1, 108.722, -149.208, 107.637, -175.657, -313.377]
  Set speed (1000.0 mm/s)
  MoveL 258 to (34.79, 183.72, 290) mm, rotated rx -90 ry -25 rz 74.51 deg; joints [-2.265, -49.571, 102.922, -142.517, 107.617, -183.579, -474.515]
  MoveL 259 to (34.79, 183.72, 290) mm, rotated rx -90 ry -25 rz 74.51 deg; joints [-2.265, -49.571, 102.922, -142.517, 107.617, -183.579, -474.515]
  Set speed (60.0 mm/s)
  MoveL 260 to (31.73, 182.3, 280) mm, rotated rx -90 ry -25 rz 72.21 deg; joints [-2.628, -49.723, 103.204, -142.729, 107.588, -183.316, -472.214]
  MoveL 261 to (27.92, 180.74, 270) mm, rotated rx -90 ry -25 rz 69.41 deg; joints [-2.992, -49.873, 103.479, -142.943, 107.558, -183.056, -469.407]
  MoveL 262 to (23.38, 179.17, 260) mm, rotated rx -90 ry -25 rz 66.13 deg; joints [-3.358, -50.019, 103.748, -143.159, 107.526, -182.797, -466.13]
  MoveL 263 to (18.11, 177.74, 250) mm, rotated rx -90 ry -25 rz 62.42 deg; joints [-3.725, -50.162, 104.011, -143.378, 107.493, -182.539, -462.417]
  MoveL 264 to (12.17, 176.57, 240) mm, rotated rx -90 ry -25 rz 58.3 deg; joints [-4.093, -50.301, 104.268, -143.599, 107.459, -182.282, -458.3]
  MoveL 265 to (5.61, 175.83, 230) mm, rotated rx -90 ry -25 rz 53.81 deg; joints [-4.463, -50.435, 104.519, -143.821, 107.424, -182.026, -453.813]
  MoveL 266 to (-1.49, 175.64, 220) mm, rotated rx -90 ry -25 rz 48.99 deg; joints [-4.834, -50.564, 104.764, -144.046, 107.389, -181.771, -448.987]
  MoveL 267 to (-9.03, 176.15, 210) mm, rotated rx -90 ry -25 rz 43.85 deg; joints [-5.207, -50.687, 105.002, -144.272, 107.355, -181.515, -443.854]
  MoveL 268 to (-16.88, 177.46, 200) mm, rotated rx -90 ry -25 rz 38.44 deg; joints [-5.581, -50.805, 105.235, -144.5, 107.322, -181.26, -438.444]
  MoveL 269 to (-24.89, 179.66, 190) mm, rotated rx -90 ry -25 rz 32.78 deg; joints [-5.956, -50.917, 105.462, -144.729, 107.289, -181.004, -432.785]
  MoveL 270 to (-32.91, 182.83, 180) mm, rotated rx -90 ry -25 rz 26.91 deg; joints [-6.332, -51.023, 105.683, -144.959, 107.258, -180.748, -426.906]
  MoveL 271 to (-40.75, 186.98, 170) mm, rotated rx -90 ry -25 rz 20.84 deg; joints [-6.709, -51.122, 105.898, -145.191, 107.229, -180.491, -420.836]
  MoveL 272 to (-48.24, 192.12, 160) mm, rotated rx -90 ry -25 rz 14.6 deg; joints [-7.088, -51.215, 106.108, -145.425, 107.201, -180.234, -414.602]
  MoveL 273 to (-55.2, 198.19, 150) mm, rotated rx -90 ry -25 rz 8.23 deg; joints [-7.468, -51.301, 106.311, -145.659, 107.174, -179.976, -408.231]
  MoveL 274 to (-61.48, 205.13, 140) mm, rotated rx -90 ry -25 rz 1.75 deg; joints [-7.849, -51.381, 106.509, -145.896, 107.149, -179.718, -401.752]
  MoveL 275 to (-66.92, 212.81, 130) mm, rotated rx -90 ry -25 rz -4.81 deg; joints [-8.231, -51.455, 106.701, -146.133, 107.124, -179.46, -395.192]
  MoveL 276 to (-71.41, 221.1, 120) mm, rotated rx -90 ry -25 rz -11.42 deg; joints [-8.614, -51.524, 106.887, -146.372, 107.101, -179.202, -388.581]
  MoveL 277 to (-74.87, 229.83, 110) mm, rotated rx -90 ry -25 rz -18.05 deg; joints [-8.998, -51.587, 107.067, -146.613, 107.077, -178.945, -381.949]
  MoveL 278 to (-77.24, 238.83, 100) mm, rotated rx -90 ry -25 rz -24.67 deg; joints [-9.383, -51.646, 107.24, -146.855, 107.054, -178.688, -375.327]
  MoveL 279 to (-78.53, 247.91, 90) mm, rotated rx -90 ry -25 rz -31.25 deg; joints [-9.769, -51.701, 107.408, -147.099, 107.029, -178.433, -368.75]
  MoveL 280 to (-78.77, 256.9, 80) mm, rotated rx -90 ry -25 rz -37.75 deg; joints [-10.156, -51.753, 107.569, -147.345, 107.003, -178.18, -362.251]
  MoveL 281 to (-78, 265.63, 70) mm, rotated rx -90 ry -25 rz -44.13 deg; joints [-10.544, -51.803, 107.724, -147.593, 106.975, -177.928, -355.868]
  MoveL 282 to (-76.35, 273.96, 60) mm, rotated rx -90 ry -25 rz -50.36 deg; joints [-10.933, -51.85, 107.873, -147.842, 106.945, -177.679, -349.641]
  MoveL 283 to (-73.92, 281.75, 50) mm, rotated rx -90 ry -25 rz -56.39 deg; joints [-11.323, -51.895, 108.015, -148.094, 106.912, -177.433, -343.608]
  MoveL 284 to (-70.87, 288.9, 40) mm, rotated rx -90 ry -25 rz -62.19 deg; joints [-11.713, -51.939, 108.151, -148.348, 106.875, -177.19, -337.812]
  MoveL 285 to (-67.34, 295.36, 30) mm, rotated rx -90 ry -25 rz -57.7 deg; joints [-12.154, -47.602, 107.647, -146.676, 118.992, -170.072, -332.296]
  MoveL 286 to (-63.51, 301.08, 20) mm, rotated rx -90 ry -25 rz -62.9 deg; joints [-12.543, -47.638, 107.767, -146.899, 118.956, -169.834, -327.105]
  MoveL 287 to (-59.54, 306.05, 10) mm, rotated rx -90 ry -25 rz -67.72 deg; joints [-12.934, -47.674, 107.881, -147.124, 118.916, -169.599, -322.281]
  MoveL 288 to (-55.59, 310.29, 0) mm, rotated rx -90 ry -25 rz -72.13 deg; joints [-13.325, -47.71, 107.988, -147.352, 118.871, -169.368, -317.87]
  Set speed (1000.0 mm/s)
  MoveL 289 to (-55.59, 310.29, 0) mm, rotated rx -90 ry -25 rz -72.13 deg; joints [-13.325, -47.71, 107.988, -147.352, 118.871, -169.368, -317.87]
  Set speed (1000.0 mm/s)
  MoveL 290 to (34.79, 183.72, 290) mm, rotated rx -90 ry -25 rz 74.51 deg; joints [-2.265, -49.571, 102.922, -142.517, 107.617, -183.579, -474.515]
  MoveL 291 to (34.79, 183.72, 290) mm, rotated rx -90 ry -25 rz 74.51 deg; joints [-2.265, -49.571, 102.922, -142.517, 107.617, -183.579, -474.515]
  Set speed (60.0 mm/s)
  MoveL 292 to (30.72, 204.12, 290) mm, rotated rx -90 ry -25 rz 78.8 deg; joints [-2.265, -48.633, 103.028, -142.309, 108.445, -182.909, -478.796]
  Set speed (1000.0 mm/s)
  MoveL 293 to (30.72, 204.12, 290) mm, rotated rx -90 ry -25 rz 78.8 deg; joints [-2.265, -48.633, 103.028, -142.309, 108.445, -182.909, -478.796]
  Set speed (1000.0 mm/s)
  MoveL 294 to (-55.59, 310.29, 0) mm, rotated rx -90 ry -25 rz -72.13 deg; joints [-13.325, -47.71, 107.988, -147.352, 118.871, -169.368, -317.87]
  MoveL 295 to (-55.59, 310.29, 0) mm, rotated rx -90 ry -25 rz -72.13 deg; joints [-13.325, -47.71, 107.988, -147.352, 118.871, -169.368, -317.87]
  Set speed (60.0 mm/s)
  MoveL 296 to (-45.21, 292.27, 0) mm, rotated rx -90 ry -25 rz -75.52 deg; joints [-13.282, -51.139, 108.719, -149.215, 107.602, -175.679, -324.484]
  Set speed (1000.0 mm/s)
  MoveL 297 to (-45.21, 292.27, 0) mm, rotated rx -90 ry -25 rz -75.52 deg; joints [-13.282, -51.139, 108.719, -149.215, 107.602, -175.679, -324.484]
  Set speed (1000.0 mm/s)
  MoveL 298 to (-55.59, 310.29, 0) mm, rotated rx -90 ry -25 rz -72.13 deg; joints [-13.325, -47.71, 107.988, -147.352, 118.871, -169.368, -317.87]
  MoveL 299 to (-55.59, 310.29, 0) mm, rotated rx -90 ry -25 rz -72.13 deg; joints [-13.325, -47.71, 107.988, -147.352, 118.871, -169.368, -317.87]
  Set speed (60.0 mm/s)
  MoveL 300 to (-59.54, 306.05, 10) mm, rotated rx -90 ry -25 rz -67.72 deg; joints [-12.934, -47.674, 107.881, -147.124, 118.916, -169.599, -322.281]
  MoveL 301 to (-63.51, 301.08, 20) mm, rotated rx -90 ry -25 rz -62.9 deg; joints [-12.543, -47.638, 107.767, -146.899, 118.956, -169.834, -327.105]
  MoveL 302 to (-67.34, 295.36, 30) mm, rotated rx -90 ry -25 rz -57.7 deg; joints [-12.154, -47.602, 107.647, -146.676, 118.992, -170.072, -332.296]
  MoveL 303 to (-70.87, 288.9, 40) mm, rotated rx -90 ry -25 rz -62.19 deg; joints [-11.713, -51.939, 108.151, -148.348, 106.875, -177.19, -337.812]
  MoveL 304 to (-73.92, 281.75, 50) mm, rotated rx -90 ry -25 rz -56.39 deg; joints [-11.323, -51.895, 108.015, -148.094, 106.912, -177.433, -343.608]
  MoveL 305 to (-76.35, 273.96, 60) mm, rotated rx -90 ry -25 rz -50.36 deg; joints [-10.933, -51.85, 107.873, -147.842, 106.945, -177.679, -349.641]
  MoveL 306 to (-78, 265.63, 70) mm, rotated rx -90 ry -25 rz -44.13 deg; joints [-10.544, -51.803, 107.724, -147.593, 106.975, -177.928, -355.868]
  MoveL 307 to (-78.77, 256.9, 80) mm, rotated rx -90 ry -25 rz -37.75 deg; joints [-10.156, -51.753, 107.569, -147.345, 107.003, -178.18, -362.251]
  MoveL 308 to (-78.53, 247.91, 90) mm, rotated rx -90 ry -25 rz -31.25 deg; joints [-9.769, -51.701, 107.408, -147.099, 107.029, -178.433, -368.75]
  MoveL 309 to (-77.24, 238.83, 100) mm, rotated rx -90 ry -25 rz -24.67 deg; joints [-9.383, -51.646, 107.24, -146.855, 107.054, -178.688, -375.327]
  MoveL 310 to (-74.87, 229.83, 110) mm, rotated rx -90 ry -25 rz -18.05 deg; joints [-8.998, -51.587, 107.067, -146.613, 107.077, -178.945, -381.949]
  MoveL 311 to (-71.41, 221.1, 120) mm, rotated rx -90 ry -25 rz -11.42 deg; joints [-8.614, -51.524, 106.887, -146.372, 107.101, -179.202, -388.581]
  MoveL 312 to (-66.92, 212.81, 130) mm, rotated rx -90 ry -25 rz -4.81 deg; joints [-8.231, -51.455, 106.701, -146.133, 107.124, -179.46, -395.192]
  MoveL 313 to (-61.48, 205.13, 140) mm, rotated rx -90 ry -25 rz 1.75 deg; joints [-7.849, -51.381, 106.509, -145.896, 107.149, -179.718, -401.752]
  MoveL 314 to (-55.2, 198.19, 150) mm, rotated rx -90 ry -25 rz 8.23 deg; joints [-7.468, -51.301, 106.311, -145.659, 107.174, -179.976, -408.231]
  MoveL 315 to (-48.24, 192.12, 160) mm, rotated rx -90 ry -25 rz 14.6 deg; joints [-7.088, -51.215, 106.108, -145.425, 107.201, -180.234, -414.602]
  MoveL 316 to (-40.75, 186.98, 170) mm, rotated rx -90 ry -25 rz 20.84 deg; joints [-6.709, -51.122, 105.898, -145.191, 107.229, -180.491, -420.836]
  MoveL 317 to (-32.91, 182.83, 180) mm, rotated rx -90 ry -25 rz 26.91 deg; joints [-6.332, -51.023, 105.683, -144.959, 107.258, -180.748, -426.906]
  MoveL 318 to (-24.89, 179.66, 190) mm, rotated rx -90 ry -25 rz 32.78 deg; joints [-5.956, -50.917, 105.462, -144.729, 107.289, -181.004, -432.785]
  MoveL 319 to (-16.88, 177.46, 200) mm, rotated rx -90 ry -25 rz 38.44 deg; joints [-5.581, -50.805, 105.235, -144.5, 107.322, -181.26, -438.444]
  MoveL 320 to (-9.03, 176.15, 210) mm, rotated rx -90 ry -25 rz 43.85 deg; joints [-5.207, -50.687, 105.002, -144.272, 107.355, -181.515, -443.854]
  MoveL 321 to (-1.49, 175.64, 220) mm, rotated rx -90 ry -25 rz 48.99 deg; joints [-4.834, -50.564, 104.764, -144.046, 107.389, -181.771, -448.987]
  MoveL 322 to (5.61, 175.83, 230) mm, rotated rx -90 ry -25 rz 53.81 deg; joints [-4.463, -50.435, 104.519, -143.821, 107.424, -182.026, -453.813]
  MoveL 323 to (12.17, 176.57, 240) mm, rotated rx -90 ry -25 rz 58.3 deg; joints [-4.093, -50.301, 104.268, -143.599, 107.459, -182.282, -458.3]
  MoveL 324 to (18.11, 177.74, 250) mm, rotated rx -90 ry -25 rz 62.42 deg; joints [-3.725, -50.162, 104.011, -143.378, 107.493, -182.539, -462.417]
  MoveL 325 to (23.38, 179.17, 260) mm, rotated rx -90 ry -25 rz 66.13 deg; joints [-3.358, -50.019, 103.748, -143.159, 107.526, -182.797, -466.13]
  MoveL 326 to (27.92, 180.74, 270) mm, rotated rx -90 ry -25 rz 69.41 deg; joints [-2.992, -49.873, 103.479, -142.943, 107.558, -183.056, -469.407]
  MoveL 327 to (31.73, 182.3, 280) mm, rotated rx -90 ry -25 rz 72.21 deg; joints [-2.628, -49.723, 103.204, -142.729, 107.588, -183.316, -472.214]
  MoveL 328 to (34.79, 183.72, 290) mm, rotated rx -90 ry -25 rz 74.51 deg; joints [-2.265, -49.571, 102.922, -142.517, 107.617, -183.579, -474.515]
  Set speed (1000.0 mm/s)
  MoveL 329 to (34.79, 183.72, 290) mm, rotated rx -90 ry -25 rz 74.51 deg; joints [-2.265, -49.571, 102.922, -142.517, 107.617, -183.579, -474.515]
  Set speed (1000.0 mm/s)
  MoveL 330 to (30.72, 204.12, 290) mm, rotated rx -90 ry -25 rz 78.8 deg; joints [-2.265, -48.633, 103.028, -142.309, 108.445, -182.909, -478.796]
  MoveL 331 to (30.72, 204.12, 290) mm, rotated rx -90 ry -25 rz 78.8 deg; joints [-2.265, -48.633, 103.028, -142.309, 108.445, -182.909, -478.796]
  Set speed (60.0 mm/s)
  MoveL 332 to (28.54, 202.85, 280) mm, rotated rx -90 ry -25 rz 76.53 deg; joints [-2.628, -48.783, 103.31, -142.522, 108.42, -182.648, -476.535]
  MoveL 333 to (25.81, 201.43, 270) mm, rotated rx -90 ry -25 rz 73.78 deg; joints [-2.992, -48.931, 103.586, -142.737, 108.394, -182.39, -473.779]
  MoveL 334 to (22.53, 199.96, 260) mm, rotated rx -90 ry -25 rz 70.56 deg; joints [-3.358, -49.077, 103.855, -142.955, 108.365, -182.133, -470.563]
  MoveL 335 to (18.7, 198.53, 250) mm, rotated rx -90 ry -25 rz 66.92 deg; joints [-3.725, -49.218, 104.119, -143.175, 108.335, -181.878, -466.921]
  MoveL 336 to (14.35, 197.26, 240) mm, rotated rx -90 ry -25 rz 62.89 deg; joints [-4.093, -49.356, 104.375, -143.397, 108.304, -181.625, -462.886]
  MoveL 337 to (9.52, 196.26, 230) mm, rotated rx -90 ry -25 rz 58.49 deg; joints [-4.463, -49.49, 104.626, -143.621, 108.272, -181.372, -458.492]
  MoveL 338 to (4.24, 195.64, 220) mm, rotated rx -90 ry -25 rz 53.77 deg; joints [-4.834, -49.618, 104.871, -143.847, 108.24, -181.12, -453.769]
  MoveL 339 to (-1.41, 195.5, 210) mm, rotated rx -90 ry -25 rz 48.75 deg; joints [-5.207, -49.742, 105.109, -144.074, 108.208, -180.869, -448.748]
  MoveL 340 to (-7.35, 195.94, 200) mm, rotated rx -90 ry -25 rz 43.46 deg; joints [-5.581, -49.86, 105.342, -144.304, 108.177, -180.617, -443.458]
  MoveL 341 to (-13.47, 197.04, 190) mm, rotated rx -90 ry -25 rz 37.93 deg; joints [-5.956, -49.972, 105.568, -144.534, 108.147, -180.365, -437.927]
  MoveL 342 to (-19.65, 198.85, 180) mm, rotated rx -90 ry -25 rz 32.18 deg; joints [-6.332, -50.078, 105.789, -144.767, 108.117, -180.113, -432.183]
  MoveL 343 to (-25.78, 201.42, 170) mm, rotated rx -90 ry -25 rz 26.25 deg; joints [-6.709, -50.177, 106.003, -145, 108.089, -179.861, -426.252]
  MoveL 344 to (-31.7, 204.73, 160) mm, rotated rx -90 ry -25 rz 20.16 deg; joints [-7.088, -50.27, 106.212, -145.235, 108.063, -179.608, -420.159]
  MoveL 345 to (-37.3, 208.79, 150) mm, rotated rx -90 ry -25 rz 13.93 deg; joints [-7.468, -50.357, 106.415, -145.472, 108.038, -179.355, -413.93]
  MoveL 346 to (-42.45, 213.53, 140) mm, rotated rx -90 ry -25 rz 7.59 deg; joints [-7.849, -50.437, 106.611, -145.709, 108.014, -179.101, -407.591]
  MoveL 347 to (-47.02, 218.88, 130) mm, rotated rx -90 ry -25 rz 1.17 deg; joints [-8.231, -50.511, 106.802, -145.949, 107.991, -178.847, -401.168]
  MoveL 348 to (-50.93, 224.75, 120) mm, rotated rx -90 ry -25 rz -5.31 deg; joints [-8.614, -50.579, 106.987, -146.189, 107.969, -178.594, -394.687]
  MoveL 349 to (-54.1, 231.02, 110) mm, rotated rx -90 ry -25 rz -11.82 deg; joints [-8.998, -50.642, 107.166, -146.431, 107.948, -178.341, -388.176]
  MoveL 350 to (-56.49, 237.56, 100) mm, rotated rx -90 ry -25 rz -18.34 deg; joints [-9.383, -50.701, 107.338, -146.675, 107.927, -178.089, -381.664]
  MoveL 351 to (-58.06, 244.24, 90) mm, rotated rx -90 ry -25 rz -24.82 deg; joints [-9.769, -50.755, 107.505, -146.92, 107.905, -177.837, -375.184]
  MoveL 352 to (-58.85, 250.92, 80) mm, rotated rx -90 ry -25 rz -31.23 deg; joints [-10.156, -50.805, 107.665, -147.168, 107.882, -177.588, -368.767]
  MoveL 353 to (-58.87, 257.48, 70) mm, rotated rx -90 ry -25 rz -37.55 deg; joints [-10.544, -50.852, 107.819, -147.417, 107.857, -177.34, -362.451]
  MoveL 354 to (-58.2, 263.79, 60) mm, rotated rx -90 ry -25 rz -43.73 deg; joints [-10.933, -50.897, 107.967, -147.667, 107.83, -177.094, -356.272]
  MoveL 355 to (-56.92, 269.76, 50) mm, rotated rx -90 ry -25 rz -49.73 deg; joints [-11.323, -50.94, 108.108, -147.92, 107.801, -176.851, -350.271]
  MoveL 356 to (-55.13, 275.3, 40) mm, rotated rx -90 ry -25 rz -55.51 deg; joints [-11.713, -50.982, 108.243, -148.175, 107.768, -176.611, -344.491]
  MoveL 357 to (-52.95, 280.35, 30) mm, rotated rx -90 ry -25 rz -61.02 deg; joints [-12.104, -51.022, 108.372, -148.432, 107.732, -176.373, -338.976]
  MoveL 358 to (-50.48, 284.87, 20) mm, rotated rx -90 ry -25 rz -66.23 deg; joints [-12.496, -51.061, 108.494, -148.691, 107.693, -176.139, -333.772]
  MoveL 359 to (-47.86, 288.84, 10) mm, rotated rx -90 ry -25 rz -71.07 deg; joints [-12.889, -51.1, 108.61, -148.952, 107.649, -175.907, -328.926]
  MoveL 360 to (-45.21, 292.27, 0) mm, rotated rx -90 ry -25 rz -75.52 deg; joints [-13.282, -51.139, 108.719, -149.215, 107.602, -175.679, -324.484]
  Set speed (1000.0 mm/s)
  MoveL 361 to (-45.21, 292.27, 0) mm, rotated rx -90 ry -25 rz -75.52 deg; joints [-13.282, -51.139, 108.719, -149.215, 107.602, -175.679, -324.484]
  Set speed (1000.0 mm/s)
  MoveL 362 to (30.72, 204.12, 290) mm, rotated rx -90 ry -25 rz 78.8 deg; joints [-2.265, -48.633, 103.028, -142.309, 108.445, -182.909, -478.796]
  MoveL 363 to (30.72, 204.12, 290) mm, rotated rx -90 ry -25 rz 78.8 deg; joints [-2.265, -48.633, 103.028, -142.309, 108.445, -182.909, -478.796]
  Set speed (60.0 mm/s)
  MoveL 364 to (58.22, 245.2, 290) mm, rotated rx -90 ry -25 rz 125.73 deg; joints [-2.265, -48.458, 103.045, -142.27, 108.596, -182.786, -525.735]
  Set speed (1000.0 mm/s)
  MoveL 365 to (58.22, 245.2, 290) mm, rotated rx -90 ry -25 rz 125.73 deg; joints [-2.265, -48.458, 103.045, -142.27, 108.596, -182.786, -525.735]
  Set speed (1000.0 mm/s)
  MoveL 366 to (-45.21, 292.27, 0) mm, rotated rx -90 ry -25 rz -75.52 deg; joints [-13.282, -51.139, 108.719, -149.215, 107.602, -175.679, -684.484]
  MoveL 367 to (-45.21, 292.27, 0) mm, rotated rx -90 ry -25 rz -75.52 deg; joints [-13.282, -51.139, 108.719, -149.215, 107.602, -175.679, -684.484]
  Set speed (60.0 mm/s)
  MoveL 368 to (-58.12, 244.54, 0) mm, rotated rx -90 ry -25 rz -25.11 deg; joints [-13.282, -51.369, 108.701, -149.255, 107.387, -175.813, -734.894]
  Set speed (1000.0 mm/s)
  MoveL 369 to (-58.12, 244.54, 0) mm, rotated rx -90 ry -25 rz -25.11 deg; joints [-13.282, -51.369, 108.701, -149.255, 107.387, -175.813, -734.894]
  Set speed (1000.0 mm/s)
  MoveL 370 to (-45.21, 292.27, 0) mm, rotated rx -90 ry -25 rz -75.52 deg; joints [-13.282, -51.139, 108.719, -149.215, 107.602, -175.679, -684.484]
  MoveL 371 to (-45.21, 292.27, 0) mm, rotated rx -90 ry -25 rz -75.52 deg; joints [-13.282, -51.139, 108.719, -149.215, 107.602, -175.679, -684.484]
  Set speed (60.0 mm/s)
  MoveL 372 to (-47.86, 288.84, 10) mm, rotated rx -90 ry -25 rz -71.07 deg; joints [-12.889, -51.1, 108.61, -148.952, 107.649, -175.907, -688.926]
  MoveL 373 to (-50.48, 284.87, 20) mm, rotated rx -90 ry -25 rz -66.23 deg; joints [-12.496, -51.061, 108.494, -148.691, 107.693, -176.139, -693.772]
  MoveL 374 to (-52.95, 280.35, 30) mm, rotated rx -90 ry -25 rz -61.02 deg; joints [-12.104, -51.022, 108.372, -148.432, 107.732, -176.373, -698.976]
  MoveL 375 to (-55.13, 275.3, 40) mm, rotated rx -90 ry -25 rz -55.51 deg; joints [-11.713, -50.982, 108.243, -148.175, 107.768, -176.611, -704.491]
  MoveL 376 to (-56.92, 269.76, 50) mm, rotated rx -90 ry -25 rz -49.73 deg; joints [-11.323, -50.94, 108.108, -147.92, 107.801, -176.851, -710.271]
  MoveL 377 to (-58.2, 263.79, 60) mm, rotated rx -90 ry -25 rz -43.73 deg; joints [-10.933, -50.897, 107.967, -147.667, 107.83, -177.094, -716.272]
  MoveL 378 to (-58.87, 257.48, 70) mm, rotated rx -90 ry -25 rz -37.55 deg; joints [-10.544, -50.852, 107.819, -147.417, 107.857, -177.34, -722.451]
  MoveL 379 to (-58.85, 250.92, 80) mm, rotated rx -90 ry -25 rz -31.23 deg; joints [-10.156, -50.805, 107.665, -147.168, 107.882, -177.588, -728.767]
  MoveL 380 to (-58.06, 244.24, 90) mm, rotated rx -90 ry -25 rz -24.82 deg; joints [-9.769, -50.755, 107.505, -146.92, 107.905, -177.837, -735.184]
  MoveL 381 to (-56.49, 237.56, 100) mm, rotated rx -90 ry -25 rz -18.34 deg; joints [-9.383, -50.701, 107.338, -146.675, 107.927, -178.089, -741.664]
  MoveL 382 to (-54.1, 231.02, 110) mm, rotated rx -90 ry -25 rz -11.82 deg; joints [-8.998, -50.642, 107.166, -146.431, 107.948, -178.341, -748.176]
  MoveL 383 to (-50.93, 224.75, 120) mm, rotated rx -90 ry -25 rz -5.31 deg; joints [-8.614, -50.579, 106.987, -146.189, 107.969, -178.594, -754.687]
  MoveL 384 to (-47.02, 218.88, 130) mm, rotated rx -90 ry -25 rz 1.17 deg; joints [-8.231, -50.511, 106.802, -145.949, 107.991, -178.847, -761.168]
  MoveL 385 to (-42.45, 213.53, 140) mm, rotated rx -90 ry -25 rz 7.59 deg; joints [-7.849, -50.437, 106.611, -145.709, 108.014, -179.101, -767.591]
  MoveL 386 to (-37.3, 208.79, 150) mm, rotated rx -90 ry -25 rz 13.93 deg; joints [-7.468, -50.357, 106.415, -145.472, 108.038, -179.355, -773.93]
  MoveL 387 to (-31.7, 204.73, 160) mm, rotated rx -90 ry -25 rz 20.16 deg; joints [-7.088, -50.27, 106.212, -145.235, 108.063, -179.608, -780.159]
  MoveL 388 to (-25.78, 201.42, 170) mm, rotated rx -90 ry -25 rz 26.25 deg; joints [-6.709, -50.177, 106.003, -145, 108.089, -179.861, -786.252]
  MoveL 389 to (-19.65, 198.85, 180) mm, rotated rx -90 ry -25 rz 32.18 deg; joints [-6.332, -50.078, 105.789, -144.767, 108.117, -180.113, -792.183]
  MoveL 390 to (-13.47, 197.04, 190) mm, rotated rx -90 ry -25 rz 37.93 deg; joints [-5.956, -49.972, 105.568, -144.534, 108.147, -180.365, -797.927]
  MoveL 391 to (-7.35, 195.94, 200) mm, rotated rx -90 ry -25 rz 43.46 deg; joints [-5.581, -49.86, 105.342, -144.304, 108.177, -180.617, -803.458]
  MoveL 392 to (-1.41, 195.5, 210) mm, rotated rx -90 ry -25 rz 48.75 deg; joints [-5.207, -49.742, 105.109, -144.074, 108.208, -180.869, -808.748]
  MoveL 393 to (4.24, 195.64, 220) mm, rotated rx -90 ry -25 rz 53.77 deg; joints [-4.834, -49.618, 104.871, -143.847, 108.24, -181.12, -813.769]
  MoveL 394 to (9.52, 196.26, 230) mm, rotated rx -90 ry -25 rz 58.49 deg; joints [-4.463, -49.49, 104.626, -143.621, 108.272, -181.372, -818.492]
  MoveL 395 to (14.35, 197.26, 240) mm, rotated rx -90 ry -25 rz 62.89 deg; joints [-4.093, -49.356, 104.375, -143.397, 108.304, -181.625, -822.886]
  MoveL 396 to (18.7, 198.53, 250) mm, rotated rx -90 ry -25 rz 66.92 deg; joints [-3.725, -49.218, 104.119, -143.175, 108.335, -181.878, -826.921]
  MoveL 397 to (22.53, 199.96, 260) mm, rotated rx -90 ry -25 rz 70.56 deg; joints [-3.358, -49.077, 103.855, -142.955, 108.365, -182.133, -830.563]
  MoveL 398 to (25.81, 201.43, 270) mm, rotated rx -90 ry -25 rz 73.78 deg; joints [-2.992, -48.931, 103.586, -142.737, 108.394, -182.39, -833.779]
  MoveL 399 to (28.54, 202.85, 280) mm, rotated rx -90 ry -25 rz 76.53 deg; joints [-2.628, -48.783, 103.31, -142.522, 108.42, -182.648, -836.535]
  MoveL 400 to (30.72, 204.12, 290) mm, rotated rx -90 ry -25 rz 78.8 deg; joints [-2.265, -48.633, 103.028, -142.309, 108.445, -182.909, -838.796]
  Set speed (1000.0 mm/s)
  MoveL 401 to (30.72, 204.12, 290) mm, rotated rx -90 ry -25 rz 78.8 deg; joints [-2.265, -48.633, 103.028, -142.309, 108.445, -182.909, -838.796]
  Set speed (1000.0 mm/s)
  MoveL 402 to (58.22, 245.2, 290) mm, rotated rx -90 ry -25 rz 125.73 deg; joints [-2.265, -48.458, 103.045, -142.27, 108.596, -182.786, -885.735]
  MoveL 403 to (58.22, 245.2, 290) mm, rotated rx -90 ry -25 rz 125.73 deg; joints [-2.265, -48.458, 103.045, -142.27, 108.596, -182.786, -885.735]
  Set speed (60.0 mm/s)
  MoveL 404 to (57.77, 242.72, 280) mm, rotated rx -90 ry -25 rz 123.34 deg; joints [-2.628, -48.614, 103.326, -142.484, 108.567, -182.529, -883.345]
  MoveL 405 to (57.08, 239.72, 270) mm, rotated rx -90 ry -25 rz 120.44 deg; joints [-2.992, -48.769, 103.601, -142.701, 108.535, -182.276, -880.439]
  MoveL 406 to (56.08, 236.26, 260) mm, rotated rx -90 ry -25 rz 117.06 deg; joints [-3.358, -48.923, 103.87, -142.921, 108.499, -182.026, -877.057]
  MoveL 407 to (54.69, 232.42, 250) mm, rotated rx -90 ry -25 rz 113.24 deg; joints [-3.725, -49.075, 104.132, -143.144, 108.461, -181.779, -873.242]
  MoveL 408 to (52.84, 228.29, 240) mm, rotated rx -90 ry -25 rz 109.03 deg; joints [-4.093, -49.225, 104.388, -143.369, 108.419, -181.535, -869.031]
  MoveL 409 to (50.46, 223.96, 230) mm, rotated rx -90 ry -25 rz 104.47 deg; joints [-4.463, -49.373, 104.637, -143.596, 108.375, -181.292, -864.466]
  MoveL 410 to (47.51, 219.54, 220) mm, rotated rx -90 ry -25 rz 99.58 deg; joints [-4.834, -49.518, 104.88, -143.825, 108.329, -181.052, -859.584]
  MoveL 411 to (43.95, 215.15, 210) mm, rotated rx -90 ry -25 rz 94.42 deg; joints [-5.207, -49.659, 105.117, -144.057, 108.282, -180.813, -854.422]
  MoveL 412 to (39.77, 210.92, 200) mm, rotated rx -90 ry -25 rz 89.02 deg; joints [-5.581, -49.797, 105.348, -144.29, 108.233, -180.575, -849.016]
  MoveL 413 to (34.96, 206.97, 190) mm, rotated rx -90 ry -25 rz 83.4 deg; joints [-5.956, -49.93, 105.572, -144.526, 108.184, -180.337, -843.399]
  MoveL 414 to (29.57, 203.44, 180) mm, rotated rx -90 ry -25 rz 77.6 deg; joints [-6.332, -50.059, 105.79, -144.763, 108.135, -180.101, -837.602]
  MoveL 415 to (23.65, 200.44, 170) mm, rotated rx -90 ry -25 rz 71.66 deg; joints [-6.709, -50.182, 106.003, -145.001, 108.086, -179.864, -831.658]
  MoveL 416 to (17.28, 198.07, 160) mm, rotated rx -90 ry -25 rz 65.59 deg; joints [-7.088, -50.299, 106.209, -145.241, 108.037, -179.627, -825.594]
  MoveL 417 to (10.57, 196.44, 150) mm, rotated rx -90 ry -25 rz 59.44 deg; joints [-7.468, -50.409, 106.41, -145.482, 107.99, -179.389, -819.438]
  MoveL 418 to (3.62, 195.59, 140) mm, rotated rx -90 ry -25 rz 53.22 deg; joints [-7.849, -50.514, 106.604, -145.725, 107.945, -179.151, -813.219]
  MoveL 419 to (-3.42, 195.58, 130) mm, rotated rx -90 ry -25 rz 46.96 deg; joints [-8.231, -50.611, 106.793, -145.968, 107.901, -178.912, -806.961]
  MoveL 420 to (-10.42, 196.41, 120) mm, rotated rx -90 ry -25 rz 40.69 deg; joints [-8.614, -50.702, 106.976, -146.213, 107.858, -178.672, -800.691]
  MoveL 421 to (-17.25, 198.06, 110) mm, rotated rx -90 ry -25 rz 34.44 deg; joints [-8.998, -50.786, 107.153, -146.459, 107.817, -178.432, -794.435]
  MoveL 422 to (-23.78, 200.49, 100) mm, rotated rx -90 ry -25 rz 28.22 deg; joints [-9.383, -50.864, 107.324, -146.706, 107.778, -178.191, -788.22]
  MoveL 423 to (-29.89, 203.62, 90) mm, rotated rx -90 ry -25 rz 22.07 deg; joints [-9.769, -50.935, 107.489, -146.955, 107.74, -177.95, -782.072]
  MoveL 424 to (-35.48, 207.36, 80) mm, rotated rx -90 ry -25 rz 16.02 deg; joints [-10.156, -51, 107.648, -147.205, 107.703, -177.709, -776.02]
  MoveL 425 to (-40.49, 211.59, 70) mm, rotated rx -90 ry -25 rz 10.09 deg; joints [-10.544, -51.06, 107.801, -147.456, 107.667, -177.468, -770.093]
  MoveL 426 to (-44.86, 216.19, 60) mm, rotated rx -90 ry -25 rz 4.32 deg; joints [-10.933, -51.115, 107.948, -147.708, 107.63, -177.227, -764.321]
  MoveL 427 to (-48.58, 221.03, 50) mm, rotated rx -90 ry -25 rz -1.26 deg; joints [-11.323, -51.165, 108.089, -147.962, 107.594, -176.987, -758.737]
  MoveL 428 to (-51.63, 225.99, 40) mm, rotated rx -90 ry -25 rz -6.62 deg; joints [-11.713, -51.212, 108.224, -148.217, 107.556, -176.749, -753.376]
  MoveL 429 to (-54.06, 230.92, 30) mm, rotated rx -90 ry -25 rz -11.73 deg; joints [-12.104, -51.255, 108.353, -148.474, 107.517, -176.512, -748.272]
  MoveL 430 to (-55.91, 235.73, 20) mm, rotated rx -90 ry -25 rz -16.54 deg; joints [-12.496, -51.295, 108.475, -148.733, 107.476, -176.277, -743.465]
  MoveL 431 to (-57.23, 240.3, 10) mm, rotated rx -90 ry -25 rz -21.01 deg; joints [-12.889, -51.333, 108.591, -148.993, 107.433, -176.044, -738.992]
  MoveL 432 to (-58.12, 244.54, 0) mm, rotated rx -90 ry -25 rz -25.11 deg; joints [-13.282, -51.369, 108.701, -149.255, 107.387, -175.813, -734.894]
  Set speed (1000.0 mm/s)
  MoveL 433 to (-58.12, 244.54, 0) mm, rotated rx -90 ry -25 rz -25.11 deg; joints [-13.282, -51.369, 108.701, -149.255, 107.387, -175.813, -734.894]
  Set speed (1000.0 mm/s)
  MoveL 434 to (58.22, 245.2, 290) mm, rotated rx -90 ry -25 rz 125.73 deg; joints [-2.265, -48.458, 103.045, -142.27, 108.596, -182.786, -885.735]
  MoveL 435 to (58.22, 245.2, 290) mm, rotated rx -90 ry -25 rz 125.73 deg; joints [-2.265, -48.458, 103.045, -142.27, 108.596, -182.786, -885.735]
  Set speed (60.0 mm/s)
  MoveL 436 to (78.63, 249.2, 290) mm, rotated rx -90 ry -25 rz 132.18 deg; joints [-2.265, -49.364, 102.948, -142.471, 107.802, -183.43, -892.181]
  Set speed (1000.0 mm/s)
  MoveL 437 to (78.63, 249.2, 290) mm, rotated rx -90 ry -25 rz 132.18 deg; joints [-2.265, -49.364, 102.948, -142.471, 107.802, -183.43, -892.181]
  Set speed (1000.0 mm/s)
  MoveL 438 to (-58.12, 244.54, 0) mm, rotated rx -90 ry -25 rz -25.11 deg; joints [-13.282, -51.369, 108.701, -149.255, 107.387, -175.813, -734.894]
  MoveL 439 to (-58.12, 244.54, 0) mm, rotated rx -90 ry -25 rz -25.11 deg; joints [-13.282, -51.369, 108.701, -149.255, 107.387, -175.813, -734.894]
  Set speed (60.0 mm/s)
  MoveL 440 to (-76.17, 234.21, 0) mm, rotated rx -90 ry -25 rz -11.3 deg; joints [-13.325, -47.995, 107.992, -147.435, 118.635, -169.541, -738.703]
  Set speed (1000.0 mm/s)
  MoveL 441 to (-76.17, 234.21, 0) mm, rotated rx -90 ry -25 rz -11.3 deg; joints [-13.325, -47.995, 107.992, -147.435, 118.635, -169.541, -738.703]
  Set speed (1000.0 mm/s)
  MoveL 442 to (-58.12, 244.54, 0) mm, rotated rx -90 ry -25 rz -25.11 deg; joints [-13.282, -51.369, 108.701, -149.255, 107.387, -175.813, -734.894]
  MoveL 443 to (-58.12, 244.54, 0) mm, rotated rx -90 ry -25 rz -25.11 deg; joints [-13.282, -51.369, 108.701, -149.255, 107.387, -175.813, -734.894]
  Set speed (60.0 mm/s)
  MoveL 444 to (-57.23, 240.3, 10) mm, rotated rx -90 ry -25 rz -21.01 deg; joints [-12.889, -51.333, 108.591, -148.993, 107.433, -176.044, -738.992]
  MoveL 445 to (-55.91, 235.73, 20) mm, rotated rx -90 ry -25 rz -16.54 deg; joints [-12.496, -51.295, 108.475, -148.733, 107.476, -176.277, -743.465]
  MoveL 446 to (-54.06, 230.92, 30) mm, rotated rx -90 ry -25 rz -11.73 deg; joints [-12.104, -51.255, 108.353, -148.474, 107.517, -176.512, -748.272]
  MoveL 447 to (-51.63, 225.99, 40) mm, rotated rx -90 ry -25 rz -6.62 deg; joints [-11.713, -51.212, 108.224, -148.217, 107.556, -176.749, -753.376]
  MoveL 448 to (-48.58, 221.03, 50) mm, rotated rx -90 ry -25 rz -1.26 deg; joints [-11.323, -51.165, 108.089, -147.962, 107.594, -176.987, -758.737]
  MoveL 449 to (-44.86, 216.19, 60) mm, rotated rx -90 ry -25 rz 4.32 deg; joints [-10.933, -51.115, 107.948, -147.708, 107.63, -177.227, -764.321]
  MoveL 450 to (-40.49, 211.59, 70) mm, rotated rx -90 ry -25 rz 10.09 deg; joints [-10.544, -51.06, 107.801, -147.456, 107.667, -177.468, -770.093]
  MoveL 451 to (-35.48, 207.36, 80) mm, rotated rx -90 ry -25 rz 16.02 deg; joints [-10.156, -51, 107.648, -147.205, 107.703, -177.709, -776.02]
  MoveL 452 to (-29.89, 203.62, 90) mm, rotated rx -90 ry -25 rz 22.07 deg; joints [-9.769, -50.935, 107.489, -146.955, 107.74, -177.95, -782.072]
  MoveL 453 to (-23.78, 200.49, 100) mm, rotated rx -90 ry -25 rz 28.22 deg; joints [-9.383, -50.864, 107.324, -146.706, 107.778, -178.191, -788.22]
  MoveL 454 to (-17.25, 198.06, 110) mm, rotated rx -90 ry -25 rz 34.44 deg; joints [-8.998, -50.786, 107.153, -146.459, 107.817, -178.432, -794.435]
  MoveL 455 to (-10.42, 196.41, 120) mm, rotated rx -90 ry -25 rz 40.69 deg; joints [-8.614, -50.702, 106.976, -146.213, 107.858, -178.672, -800.691]
  MoveL 456 to (-3.42, 195.58, 130) mm, rotated rx -90 ry -25 rz 46.96 deg; joints [-8.231, -50.611, 106.793, -145.968, 107.901, -178.912, -806.961]
  MoveL 457 to (3.62, 195.59, 140) mm, rotated rx -90 ry -25 rz 53.22 deg; joints [-7.849, -50.514, 106.604, -145.725, 107.945, -179.151, -813.219]
  MoveL 458 to (10.57, 196.44, 150) mm, rotated rx -90 ry -25 rz 59.44 deg; joints [-7.468, -50.409, 106.41, -145.482, 107.99, -179.389, -819.438]
  MoveL 459 to (17.28, 198.07, 160) mm, rotated rx -90 ry -25 rz 65.59 deg; joints [-7.088, -50.299, 106.209, -145.241, 108.037, -179.627, -825.594]
  MoveL 460 to (23.65, 200.44, 170) mm, rotated rx -90 ry -25 rz 71.66 deg; joints [-6.709, -50.182, 106.003, -145.001, 108.086, -179.864, -831.658]
  MoveL 461 to (29.57, 203.44, 180) mm, rotated rx -90 ry -25 rz 77.6 deg; joints [-6.332, -50.059, 105.79, -144.763, 108.135, -180.101, -837.602]
  MoveL 462 to (34.96, 206.97, 190) mm, rotated rx -90 ry -25 rz 83.4 deg; joints [-5.956, -49.93, 105.572, -144.526, 108.184, -180.337, -843.399]
  MoveL 463 to (39.77, 210.92, 200) mm, rotated rx -90 ry -25 rz 89.02 deg; joints [-5.581, -49.797, 105.348, -144.29, 108.233, -180.575, -849.016]
  MoveL 464 to (43.95, 215.15, 210) mm, rotated rx -90 ry -25 rz 94.42 deg; joints [-5.207, -49.659, 105.117, -144.057, 108.282, -180.813, -854.422]
  MoveL 465 to (47.51, 219.54, 220) mm, rotated rx -90 ry -25 rz 99.58 deg; joints [-4.834, -49.518, 104.88, -143.825, 108.329, -181.052, -859.584]
  MoveL 466 to (50.46, 223.96, 230) mm, rotated rx -90 ry -25 rz 104.47 deg; joints [-4.463, -49.373, 104.637, -143.596, 108.375, -181.292, -864.466]
  MoveL 467 to (52.84, 228.29, 240) mm, rotated rx -90 ry -25 rz 109.03 deg; joints [-4.093, -49.225, 104.388, -143.369, 108.419, -181.535, -869.031]
  MoveL 468 to (54.69, 232.42, 250) mm, rotated rx -90 ry -25 rz 113.24 deg; joints [-3.725, -49.075, 104.132, -143.144, 108.461, -181.779, -873.242]
  MoveL 469 to (56.08, 236.26, 260) mm, rotated rx -90 ry -25 rz 117.06 deg; joints [-3.358, -48.923, 103.87, -142.921, 108.499, -182.026, -877.057]
  MoveL 470 to (57.08, 239.72, 270) mm, rotated rx -90 ry -25 rz 120.44 deg; joints [-2.992, -48.769, 103.601, -142.701, 108.535, -182.276, -880.439]
  MoveL 471 to (57.77, 242.72, 280) mm, rotated rx -90 ry -25 rz 123.34 deg; joints [-2.628, -48.614, 103.326, -142.484, 108.567, -182.529, -883.345]
  MoveL 472 to (58.22, 245.2, 290) mm, rotated rx -90 ry -25 rz 125.73 deg; joints [-2.265, -48.458, 103.045, -142.27, 108.596, -182.786, -885.735]
  Set speed (1000.0 mm/s)
  MoveL 473 to (58.22, 245.2, 290) mm, rotated rx -90 ry -25 rz 125.73 deg; joints [-2.265, -48.458, 103.045, -142.27, 108.596, -182.786, -885.735]
  Set speed (1000.0 mm/s)
  MoveL 474 to (78.63, 249.2, 290) mm, rotated rx -90 ry -25 rz 132.18 deg; joints [-2.265, -49.364, 102.948, -142.471, 107.802, -183.43, -892.181]
  MoveL 475 to (78.63, 249.2, 290) mm, rotated rx -90 ry -25 rz 132.18 deg; joints [-2.265, -49.364, 102.948, -142.471, 107.802, -183.43, -892.181]
  Set speed (60.0 mm/s)
  MoveL 476 to (78.34, 245.85, 280) mm, rotated rx -90 ry -25 rz 129.76 deg; joints [-2.628, -49.522, 103.229, -142.685, 107.769, -183.172, -889.758]
  MoveL 477 to (77.78, 241.77, 270) mm, rotated rx -90 ry -25 rz 126.81 deg; joints [-2.992, -49.68, 103.504, -142.901, 107.732, -182.918, -886.809]
  MoveL 478 to (76.86, 237.05, 260) mm, rotated rx -90 ry -25 rz 123.37 deg; joints [-3.358, -49.836, 103.772, -143.12, 107.691, -182.666, -883.374]
  MoveL 479 to (75.48, 231.77, 250) mm, rotated rx -90 ry -25 rz 119.49 deg; joints [-3.725, -49.991, 104.033, -143.342, 107.648, -182.418, -879.493]
  MoveL 480 to (73.51, 226.04, 240) mm, rotated rx -90 ry -25 rz 115.21 deg; joints [-4.093, -50.144, 104.288, -143.566, 107.601, -182.172, -875.208]
  MoveL 481 to (70.88, 219.99, 230) mm, rotated rx -90 ry -25 rz 110.56 deg; joints [-4.463, -50.295, 104.537, -143.792, 107.551, -181.929, -870.555]
  MoveL 482 to (67.49, 213.75, 220) mm, rotated rx -90 ry -25 rz 105.58 deg; joints [-4.834, -50.443, 104.779, -144.021, 107.499, -181.687, -865.575]
  MoveL 483 to (63.28, 207.47, 210) mm, rotated rx -90 ry -25 rz 100.31 deg; joints [-5.207, -50.588, 105.015, -144.251, 107.446, -181.447, -860.305]
  MoveL 484 to (58.22, 201.33, 200) mm, rotated rx -90 ry -25 rz 94.78 deg; joints [-5.581, -50.73, 105.245, -144.484, 107.391, -181.208, -854.781]
  MoveL 485 to (52.31, 195.49, 190) mm, rotated rx -90 ry -25 rz 89.04 deg; joints [-5.956, -50.867, 105.469, -144.719, 107.336, -180.97, -849.037]
  MoveL 486 to (45.56, 190.13, 180) mm, rotated rx -90 ry -25 rz 83.11 deg; joints [-6.332, -51, 105.686, -144.955, 107.28, -180.732, -843.107]
  MoveL 487 to (38.04, 185.42, 170) mm, rotated rx -90 ry -25 rz 77.02 deg; joints [-6.709, -51.127, 105.898, -145.192, 107.224, -180.494, -837.024]
  MoveL 488 to (29.85, 181.5, 160) mm, rotated rx -90 ry -25 rz 70.82 deg; joints [-7.088, -51.248, 106.104, -145.431, 107.169, -180.256, -830.818]
  MoveL 489 to (21.11, 178.51, 150) mm, rotated rx -90 ry -25 rz 64.52 deg; joints [-7.468, -51.364, 106.303, -145.672, 107.116, -180.018, -824.519]
  MoveL 490 to (11.96, 176.54, 140) mm, rotated rx -90 ry -25 rz 58.16 deg; joints [-7.849, -51.472, 106.497, -145.913, 107.063, -179.779, -818.157]
  MoveL 491 to (2.59, 175.67, 130) mm, rotated rx -90 ry -25 rz 51.76 deg; joints [-8.231, -51.575, 106.686, -146.156, 107.012, -179.538, -811.758]
  MoveL 492 to (-6.83, 175.92, 120) mm, rotated rx -90 ry -25 rz 45.35 deg; joints [-8.614, -51.67, 106.868, -146.4, 106.963, -179.297, -805.352]
  MoveL 493 to (-16.13, 177.3, 110) mm, rotated rx -90 ry -25 rz 38.97 deg; joints [-8.998, -51.758, 107.045, -146.645, 106.916, -179.056, -798.967]
  MoveL 494 to (-25.11, 179.73, 100) mm, rotated rx -90 ry -25 rz 42.63 deg; joints [-9.449, -47.524, 106.634, -145.263, 118.984, -171.968, -792.629]
  MoveL 495 to (-33.62, 183.16, 90) mm, rotated rx -90 ry -25 rz 36.37 deg; joints [-9.833, -47.593, 106.798, -145.472, 118.951, -171.721, -786.369]
  MoveL 496 to (-41.52, 187.45, 80) mm, rotated rx -90 ry -25 rz 30.21 deg; joints [-10.217, -47.655, 106.955, -145.683, 118.918, -171.474, -780.214]
  MoveL 497 to (-48.7, 192.48, 70) mm, rotated rx -90 ry -25 rz 24.2 deg; joints [-10.603, -47.711, 107.107, -145.896, 118.886, -171.227, -774.197]
  MoveL 498 to (-55.08, 198.08, 60) mm, rotated rx -90 ry -25 rz 18.35 deg; joints [-10.989, -47.762, 107.252, -146.11, 118.854, -170.981, -768.347]
  MoveL 499 to (-60.61, 204.07, 50) mm, rotated rx -90 ry -25 rz 12.7 deg; joints [-11.377, -47.809, 107.391, -146.326, 118.822, -170.736, -762.698]
  MoveL 500 to (-65.29, 210.3, 40) mm, rotated rx -90 ry -25 rz 7.28 deg; joints [-11.765, -47.852, 107.524, -146.543, 118.788, -170.493, -757.284]
  MoveL 501 to (-69.12, 216.58, 30) mm, rotated rx -90 ry -25 rz 2.14 deg; joints [-12.154, -47.891, 107.65, -146.763, 118.753, -170.251, -752.14]
  MoveL 502 to (-72.16, 222.75, 20) mm, rotated rx -90 ry -25 rz -2.7 deg; joints [-12.543, -47.928, 107.77, -146.985, 118.716, -170.012, -747.303]
  MoveL 503 to (-74.48, 228.68, 10) mm, rotated rx -90 ry -25 rz -7.19 deg; joints [-12.934, -47.962, 107.884, -147.208, 118.677, -169.775, -742.811]
  MoveL 504 to (-76.17, 234.21, 0) mm, rotated rx -90 ry -25 rz -11.3 deg; joints [-13.325, -47.995, 107.992, -147.435, 118.635, -169.541, -738.703]
  Set speed (1000.0 mm/s)
  MoveL 505 to (-76.17, 234.21, 0) mm, rotated rx -90 ry -25 rz -11.3 deg; joints [-13.325, -47.995, 107.992, -147.435, 118.635, -169.541, -738.703]
  Set speed (1000.0 mm/s)
  MoveL 506 to (78.63, 249.2, 290) mm, rotated rx -90 ry -25 rz 132.18 deg; joints [-2.265, -49.364, 102.948, -142.471, 107.802, -183.43, -892.181]
  MoveL 507 to (78.63, 249.2, 290) mm, rotated rx -90 ry -25 rz 132.18 deg; joints [-2.265, -49.364, 102.948, -142.471, 107.802, -183.43, -892.181]
  Set speed (60.0 mm/s)
  MoveL 508 to (58.93, 255.88, 290) mm, rotated rx -90 ry -25 rz 136 deg; joints [-2.265, -48.411, 103.049, -142.26, 108.636, -182.753, -895.998]
  Set speed (1000.0 mm/s)
  MoveL 509 to (58.93, 255.88, 290) mm, rotated rx -90 ry -25 rz 136 deg; joints [-2.265, -48.411, 103.049, -142.26, 108.636, -182.753, -895.998]
  Set speed (1000.0 mm/s)
  MoveL 510 to (-76.17, 234.21, 0) mm, rotated rx -90 ry -25 rz -11.3 deg; joints [-13.325, -47.995, 107.992, -147.435, 118.635, -169.541, -738.703]
  MoveL 511 to (-76.17, 234.21, 0) mm, rotated rx -90 ry -25 rz -11.3 deg; joints [-13.325, -47.995, 107.992, -147.435, 118.635, -169.541, -738.703]
  Set speed (60.0 mm/s)
  MoveL 512 to (-55.37, 234.2, 0) mm, rotated rx -90 ry -25 rz -15.01 deg; joints [-13.282, -51.417, 108.696, -149.263, 107.343, -175.84, -744.986]
  Set speed (1000.0 mm/s)
  MoveL 513 to (-55.37, 234.2, 0) mm, rotated rx -90 ry -25 rz -15.01 deg; joints [-13.282, -51.417, 108.696, -149.263, 107.343, -175.84, -744.986]
  Set speed (1000.0 mm/s)
  MoveL 514 to (-76.17, 234.21, 0) mm, rotated rx -90 ry -25 rz -11.3 deg; joints [-13.325, -47.995, 107.992, -147.435, 118.635, -169.541, -738.703]
  MoveL 515 to (-76.17, 234.21, 0) mm, rotated rx -90 ry -25 rz -11.3 deg; joints [-13.325, -47.995, 107.992, -147.435, 118.635, -169.541, -738.703]
  Set speed (60.0 mm/s)
  MoveL 516 to (-74.48, 228.68, 10) mm, rotated rx -90 ry -25 rz -7.19 deg; joints [-12.934, -47.962, 107.884, -147.208, 118.677, -169.775, -742.811]
  MoveL 517 to (-72.16, 222.75, 20) mm, rotated rx -90 ry -25 rz -2.7 deg; joints [-12.543, -47.928, 107.77, -146.985, 118.716, -170.012, -747.303]
  MoveL 518 to (-69.12, 216.58, 30) mm, rotated rx -90 ry -25 rz 2.14 deg; joints [-12.154, -47.891, 107.65, -146.763, 118.753, -170.251, -752.14]
  MoveL 519 to (-65.29, 210.3, 40) mm, rotated rx -90 ry -25 rz 7.28 deg; joints [-11.765, -47.852, 107.524, -146.543, 118.788, -170.493, -757.284]
  MoveL 520 to (-60.61, 204.07, 50) mm, rotated rx -90 ry -25 rz 12.7 deg; joints [-11.377, -47.809, 107.391, -146.326, 118.822, -170.736, -762.698]
  MoveL 521 to (-55.08, 198.08, 60) mm, rotated rx -90 ry -25 rz 18.35 deg; joints [-10.989, -47.762, 107.252, -146.11, 118.854, -170.981, -768.347]
  MoveL 522 to (-48.7, 192.48, 70) mm, rotated rx -90 ry -25 rz 24.2 deg; joints [-10.603, -47.711, 107.107, -145.896, 118.886, -171.227, -774.197]
  MoveL 523 to (-41.52, 187.45, 80) mm, rotated rx -90 ry -25 rz 30.21 deg; joints [-10.217, -47.655, 106.955, -145.683, 118.918, -171.474, -780.214]
  MoveL 524 to (-33.62, 183.16, 90) mm, rotated rx -90 ry -25 rz 36.37 deg; joints [-9.833, -47.593, 106.798, -145.472, 118.951, -171.721, -786.369]
  MoveL 525 to (-25.11, 179.73, 100) mm, rotated rx -90 ry -25 rz 42.63 deg; joints [-9.449, -47.524, 106.634, -145.263, 118.984, -171.968, -792.629]
  MoveL 526 to (-16.13, 177.3, 110) mm, rotated rx -90 ry -25 rz 38.97 deg; joints [-8.998, -51.758, 107.045, -146.645, 106.916, -179.056, -798.967]
  MoveL 527 to (-6.83, 175.92, 120) mm, rotated rx -90 ry -25 rz 45.35 deg; joints [-8.614, -51.67, 106.868, -146.4, 106.963, -179.297, -805.352]
  MoveL 528 to (2.59, 175.67, 130) mm, rotated rx -90 ry -25 rz 51.76 deg; joints [-8.231, -51.575, 106.686, -146.156, 107.012, -179.538, -811.758]
  MoveL 529 to (11.96, 176.54, 140) mm, rotated rx -90 ry -25 rz 58.16 deg; joints [-7.849, -51.472, 106.497, -145.913, 107.063, -179.779, -818.157]
  MoveL 530 to (21.11, 178.51, 150) mm, rotated rx -90 ry -25 rz 64.52 deg; joints [-7.468, -51.364, 106.303, -145.672, 107.116, -180.018, -824.519]
  MoveL 531 to (29.85, 181.5, 160) mm, rotated rx -90 ry -25 rz 70.82 deg; joints [-7.088, -51.248, 106.104, -145.431, 107.169, -180.256, -830.818]
  MoveL 532 to (38.04, 185.42, 170) mm, rotated rx -90 ry -25 rz 77.02 deg; joints [-6.709, -51.127, 105.898, -145.192, 107.224, -180.494, -837.024]
  MoveL 533 to (45.56, 190.13, 180) mm, rotated rx -90 ry -25 rz 83.11 deg; joints [-6.332, -51, 105.686, -144.955, 107.28, -180.732, -843.107]
  MoveL 534 to (52.31, 195.49, 190) mm, rotated rx -90 ry -25 rz 89.04 deg; joints [-5.956, -50.867, 105.469, -144.719, 107.336, -180.97, -849.037]
  MoveL 535 to (58.22, 201.33, 200) mm, rotated rx -90 ry -25 rz 94.78 deg; joints [-5.581, -50.73, 105.245, -144.484, 107.391, -181.208, -854.781]
  MoveL 536 to (63.28, 207.47, 210) mm, rotated rx -90 ry -25 rz 100.31 deg; joints [-5.207, -50.588, 105.015, -144.251, 107.446, -181.447, -860.305]
  MoveL 537 to (67.49, 213.75, 220) mm, rotated rx -90 ry -25 rz 105.58 deg; joints [-4.834, -50.443, 104.779, -144.021, 107.499, -181.687, -865.575]
  MoveL 538 to (70.88, 219.99, 230) mm, rotated rx -90 ry -25 rz 110.56 deg; joints [-4.463, -50.295, 104.537, -143.792, 107.551, -181.929, -870.555]
  MoveL 539 to (73.51, 226.04, 240) mm, rotated rx -90 ry -25 rz 115.21 deg; joints [-4.093, -50.144, 104.288, -143.566, 107.601, -182.172, -875.208]
  MoveL 540 to (75.48, 231.77, 250) mm, rotated rx -90 ry -25 rz 119.49 deg; joints [-3.725, -49.991, 104.033, -143.342, 107.648, -182.418, -879.493]
  MoveL 541 to (76.86, 237.05, 260) mm, rotated rx -90 ry -25 rz 123.37 deg; joints [-3.358, -49.836, 103.772, -143.12, 107.691, -182.666, -883.374]
  MoveL 542 to (77.78, 241.77, 270) mm, rotated rx -90 ry -25 rz 126.81 deg; joints [-2.992, -49.68, 103.504, -142.901, 107.732, -182.918, -886.809]
  MoveL 543 to (78.34, 245.85, 280) mm, rotated rx -90 ry -25 rz 129.76 deg; joints [-2.628, -49.522, 103.229, -142.685, 107.769, -183.172, -889.758]
  MoveL 544 to (78.63, 249.2, 290) mm, rotated rx -90 ry -25 rz 132.18 deg; joints [-2.265, -49.364, 102.948, -142.471, 107.802, -183.43, -892.181]
  Set speed (1000.0 mm/s)
  MoveL 545 to (78.63, 249.2, 290) mm, rotated rx -90 ry -25 rz 132.18 deg; joints [-2.265, -49.364, 102.948, -142.471, 107.802, -183.43, -892.181]
  Set speed (1000.0 mm/s)
  MoveL 546 to (58.93, 255.88, 290) mm, rotated rx -90 ry -25 rz 136 deg; joints [-2.265, -48.411, 103.049, -142.26, 108.636, -182.753, -895.998]
  MoveL 547 to (58.93, 255.88, 290) mm, rotated rx -90 ry -25 rz 136 deg; joints [-2.265, -48.411, 103.049, -142.26, 108.636, -182.753, -895.998]
  Set speed (60.0 mm/s)
  MoveL 548 to (58.94, 253.36, 280) mm, rotated rx -90 ry -25 rz 133.57 deg; joints [-2.628, -48.567, 103.33, -142.474, 108.608, -182.497, -893.568]
  MoveL 549 to (58.8, 250.28, 270) mm, rotated rx -90 ry -25 rz 130.62 deg; joints [-2.992, -48.722, 103.605, -142.691, 108.575, -182.244, -890.615]
  MoveL 550 to (58.44, 246.7, 260) mm, rotated rx -90 ry -25 rz 127.18 deg; joints [-3.358, -48.877, 103.874, -142.911, 108.539, -181.995, -887.181]
  MoveL 551 to (57.77, 242.68, 250) mm, rotated rx -90 ry -25 rz 123.31 deg; joints [-3.725, -49.03, 104.136, -143.134, 108.5, -181.748, -883.306]
  MoveL 552 to (56.69, 238.28, 240) mm, rotated rx -90 ry -25 rz 119.03 deg; joints [-4.093, -49.181, 104.391, -143.359, 108.457, -181.505, -879.034]
  MoveL 553 to (55.14, 233.59, 230) mm, rotated rx -90 ry -25 rz 114.41 deg; joints [-4.463, -49.331, 104.641, -143.587, 108.412, -181.264, -874.405]
  MoveL 554 to (53.04, 228.71, 220) mm, rotated rx -90 ry -25 rz 109.46 deg; joints [-4.834, -49.478, 104.884, -143.817, 108.364, -181.025, -869.46]
  MoveL 555 to (50.33, 223.75, 210) mm, rotated rx -90 ry -25 rz 104.24 deg; joints [-5.207, -49.622, 105.12, -144.049, 108.314, -180.788, -864.235]
  MoveL 556 to (46.98, 218.83, 200) mm, rotated rx -90 ry -25 rz 98.77 deg; joints [-5.581, -49.763, 105.351, -144.283, 108.263, -180.552, -858.769]
  MoveL 557 to (42.97, 214.08, 190) mm, rotated rx -90 ry -25 rz 93.1 deg; joints [-5.956, -49.9, 105.575, -144.519, 108.211, -180.317, -853.096]
  MoveL 558 to (38.31, 209.62, 180) mm, rotated rx -90 ry -25 rz 87.25 deg; joints [-6.332, -50.032, 105.793, -144.757, 108.158, -180.083, -847.251]
  MoveL 559 to (33.03, 205.6, 170) mm, rotated rx -90 ry -25 rz 81.26 deg; joints [-6.709, -50.16, 106.005, -144.997, 108.105, -179.849, -841.263]
  MoveL 560 to (27.19, 202.13, 160) mm, rotated rx -90 ry -25 rz 75.16 deg; joints [-7.088, -50.281, 106.211, -145.237, 108.053, -179.615, -835.164]
  MoveL 561 to (20.88, 199.3, 150) mm, rotated rx -90 ry -25 rz 68.98 deg; joints [-7.468, -50.397, 106.411, -145.48, 108.001, -179.381, -828.983]
  MoveL 562 to (14.2, 197.22, 140) mm, rotated rx -90 ry -25 rz 62.75 deg; joints [-7.849, -50.507, 106.605, -145.723, 107.951, -179.146, -822.746]
  MoveL 563 to (7.28, 195.93, 130) mm, rotated rx -90 ry -25 rz 56.48 deg; joints [-8.231, -50.61, 106.793, -145.968, 107.902, -178.911, -816.481]
  MoveL 564 to (0.24, 195.48, 120) mm, rotated rx -90 ry -25 rz 50.21 deg; joints [-8.614, -50.706, 106.976, -146.214, 107.855, -178.675, -810.213]
  MoveL 565 to (-6.77, 195.87, 110) mm, rotated rx -90 ry -25 rz 43.97 deg; joints [-8.998, -50.795, 107.152, -146.461, 107.809, -178.438, -803.969]
  MoveL 566 to (-13.63, 197.08, 100) mm, rotated rx -90 ry -25 rz 37.78 deg; joints [-9.383, -50.878, 107.322, -146.709, 107.765, -178.2, -797.775]
  MoveL 567 to (-20.21, 199.05, 90) mm, rotated rx -90 ry -25 rz 31.66 deg; joints [-9.769, -50.954, 107.487, -146.959, 107.722, -177.962, -791.658]
  MoveL 568 to (-26.38, 201.72, 80) mm, rotated rx -90 ry -25 rz 25.64 deg; joints [-10.156, -51.025, 107.646, -147.209, 107.681, -177.724, -785.644]
  MoveL 569 to (-32.08, 204.97, 70) mm, rotated rx -90 ry -25 rz 19.76 deg; joints [-10.544, -51.089, 107.799, -147.461, 107.64, -177.485, -779.763]
  MoveL 570 to (-37.21, 208.71, 60) mm, rotated rx -90 ry -25 rz 14.04 deg; joints [-10.933, -51.148, 107.945, -147.714, 107.6, -177.247, -774.043]
  MoveL 571 to (-41.73, 212.8, 50) mm, rotated rx -90 ry -25 rz 8.52 deg; joints [-11.323, -51.202, 108.086, -147.968, 107.56, -177.009, -768.517]
  MoveL 572 to (-45.64, 217.12, 40) mm, rotated rx -90 ry -25 rz 3.22 deg; joints [-11.713, -51.251, 108.22, -148.224, 107.52, -176.773, -763.217]
  MoveL 573 to (-48.92, 221.54, 30) mm, rotated rx -90 ry -25 rz -1.82 deg; joints [-12.104, -51.297, 108.349, -148.482, 107.478, -176.537, -758.176]
  MoveL 574 to (-51.6, 225.93, 20) mm, rotated rx -90 ry -25 rz -6.57 deg; joints [-12.496, -51.34, 108.471, -148.74, 107.435, -176.303, -753.433]
  MoveL 575 to (-53.73, 230.19, 10) mm, rotated rx -90 ry -25 rz -10.98 deg; joints [-12.889, -51.379, 108.587, -149.001, 107.39, -176.071, -749.023]
  MoveL 576 to (-55.37, 234.2, 0) mm, rotated rx -90 ry -25 rz -15.01 deg; joints [-13.282, -51.417, 108.696, -149.263, 107.343, -175.84, -744.986]
  Set speed (1000.0 mm/s)
  MoveL 577 to (-55.37, 234.2, 0) mm, rotated rx -90 ry -25 rz -15.01 deg; joints [-13.282, -51.417, 108.696, -149.263, 107.343, -175.84, -744.986]
  Set speed (1000.0 mm/s)
  MoveL 578 to (58.93, 255.88, 290) mm, rotated rx -90 ry -25 rz 136 deg; joints [-2.265, -48.411, 103.049, -142.26, 108.636, -182.753, -895.998]
  MoveL 579 to (58.93, 255.88, 290) mm, rotated rx -90 ry -25 rz 136 deg; joints [-2.265, -48.411, 103.049, -142.26, 108.636, -182.753, -895.998]
  Set speed (60.0 mm/s)
  MoveL 580 to (37.11, 300.24, 290) mm, rotated rx -90 ry -25 rz -172.69 deg; joints [-2.265, -48.205, 103.066, -142.213, 108.813, -182.608, -947.315]
  Set speed (1000.0 mm/s)
  MoveL 581 to (37.11, 300.24, 290) mm, rotated rx -90 ry -25 rz -172.69 deg; joints [-2.265, -48.205, 103.066, -142.213, 108.813, -182.608, -947.315]
  Set speed (1000.0 mm/s)
  MoveL 582 to (-55.37, 234.2, 0) mm, rotated rx -90 ry -25 rz -15.01 deg; joints [-13.282, -51.417, 108.696, -149.263, 107.343, -175.84, -1104.986]
  MoveL 583 to (-55.37, 234.2, 0) mm, rotated rx -90 ry -25 rz -15.01 deg; joints [-13.282, -51.417, 108.696, -149.263, 107.343, -175.84, -1104.986]
  Set speed (60.0 mm/s)
  MoveL 584 to (-20.49, 199.16, 0) mm, rotated rx -90 ry -25 rz 31.39 deg; joints [-13.282, -51.572, 108.683, -149.29, 107.197, -175.931, -1151.385]
  Set speed (1000.0 mm/s)
  MoveL 585 to (-20.49, 199.16, 0) mm, rotated rx -90 ry -25 rz 31.39 deg; joints [-13.282, -51.572, 108.683, -149.29, 107.197, -175.931, -1151.385]
  Set speed (1000.0 mm/s)
  MoveL 586 to (-55.37, 234.2, 0) mm, rotated rx -90 ry -25 rz -15.01 deg; joints [-13.282, -51.417, 108.696, -149.263, 107.343, -175.84, -1104.986]
  MoveL 587 to (-55.37, 234.2, 0) mm, rotated rx -90 ry -25 rz -15.01 deg; joints [-13.282, -51.417, 108.696, -149.263, 107.343, -175.84, -1104.986]
  Set speed (60.0 mm/s)
  MoveL 588 to (-53.73, 230.19, 10) mm, rotated rx -90 ry -25 rz -10.98 deg; joints [-12.889, -51.379, 108.587, -149.001, 107.39, -176.071, -1109.023]
  MoveL 589 to (-51.6, 225.93, 20) mm, rotated rx -90 ry -25 rz -6.57 deg; joints [-12.496, -51.34, 108.471, -148.74, 107.435, -176.303, -1113.433]
  MoveL 590 to (-48.92, 221.54, 30) mm, rotated rx -90 ry -25 rz -1.82 deg; joints [-12.104, -51.297, 108.349, -148.482, 107.478, -176.537, -1118.176]
  MoveL 591 to (-45.64, 217.12, 40) mm, rotated rx -90 ry -25 rz 3.22 deg; joints [-11.713, -51.251, 108.22, -148.224, 107.52, -176.773, -1123.217]
  MoveL 592 to (-41.73, 212.8, 50) mm, rotated rx -90 ry -25 rz 8.52 deg; joints [-11.323, -51.202, 108.086, -147.968, 107.56, -177.009, -1128.517]
  MoveL 593 to (-37.21, 208.71, 60) mm, rotated rx -90 ry -25 rz 14.04 deg; joints [-10.933, -51.148, 107.945, -147.714, 107.6, -177.247, -1134.043]
  MoveL 594 to (-32.08, 204.97, 70) mm, rotated rx -90 ry -25 rz 19.76 deg; joints [-10.544, -51.089, 107.799, -147.461, 107.64, -177.485, -1139.763]
  MoveL 595 to (-26.38, 201.72, 80) mm, rotated rx -90 ry -25 rz 25.64 deg; joints [-10.156, -51.025, 107.646, -147.209, 107.681, -177.724, -1145.644]
  MoveL 596 to (-20.21, 199.05, 90) mm, rotated rx -90 ry -25 rz 31.66 deg; joints [-9.769, -50.954, 107.487, -146.959, 107.722, -177.962, -1151.658]
  MoveL 597 to (-13.63, 197.08, 100) mm, rotated rx -90 ry -25 rz 37.78 deg; joints [-9.383, -50.878, 107.322, -146.709, 107.765, -178.2, -1157.775]
  MoveL 598 to (-6.77, 195.87, 110) mm, rotated rx -90 ry -25 rz 43.97 deg; joints [-8.998, -50.795, 107.152, -146.461, 107.809, -178.438, -1163.969]
  MoveL 599 to (0.24, 195.48, 120) mm, rotated rx -90 ry -25 rz 50.21 deg; joints [-8.614, -50.706, 106.976, -146.214, 107.855, -178.675, -1170.213]
  MoveL 600 to (7.28, 195.93, 130) mm, rotated rx -90 ry -25 rz 56.48 deg; joints [-8.231, -50.61, 106.793, -145.968, 107.902, -178.911, -1176.481]
  MoveL 601 to (14.2, 197.22, 140) mm, rotated rx -90 ry -25 rz 62.75 deg; joints [-7.849, -50.507, 106.605, -145.723, 107.951, -179.146, -1182.746]
  MoveL 602 to (20.88, 199.3, 150) mm, rotated rx -90 ry -25 rz 68.98 deg; joints [-7.468, -50.397, 106.411, -145.48, 108.001, -179.381, -1188.983]
  MoveL 603 to (27.19, 202.13, 160) mm, rotated rx -90 ry -25 rz 75.16 deg; joints [-7.088, -50.281, 106.211, -145.237, 108.053, -179.615, -1195.164]
  MoveL 604 to (33.03, 205.6, 170) mm, rotated rx -90 ry -25 rz 81.26 deg; joints [-6.709, -50.16, 106.005, -144.997, 108.105, -179.849, -1201.263]
  MoveL 605 to (38.31, 209.62, 180) mm, rotated rx -90 ry -25 rz 87.25 deg; joints [-6.332, -50.032, 105.793, -144.757, 108.158, -180.083, -1207.251]
  MoveL 606 to (42.97, 214.08, 190) mm, rotated rx -90 ry -25 rz 93.1 deg; joints [-5.956, -49.9, 105.575, -144.519, 108.211, -180.317, -1213.096]
  MoveL 607 to (46.98, 218.83, 200) mm, rotated rx -90 ry -25 rz 98.77 deg; joints [-5.581, -49.763, 105.351, -144.283, 108.263, -180.552, -1218.769]
  MoveL 608 to (50.33, 223.75, 210) mm, rotated rx -90 ry -25 rz 104.24 deg; joints [-5.207, -49.622, 105.12, -144.049, 108.314, -180.788, -1224.235]
  MoveL 609 to (53.04, 228.71, 220) mm, rotated rx -90 ry -25 rz 109.46 deg; joints [-4.834, -49.478, 104.884, -143.817, 108.364, -181.025, -1229.46]
  MoveL 610 to (55.14, 233.59, 230) mm, rotated rx -90 ry -25 rz 114.41 deg; joints [-4.463, -49.331, 104.641, -143.587, 108.412, -181.264, -1234.405]
  MoveL 611 to (56.69, 238.28, 240) mm, rotated rx -90 ry -25 rz 119.03 deg; joints [-4.093, -49.181, 104.391, -143.359, 108.457, -181.505, -1239.034]
  MoveL 612 to (57.77, 242.68, 250) mm, rotated rx -90 ry -25 rz 123.31 deg; joints [-3.725, -49.03, 104.136, -143.134, 108.5, -181.748, -1243.306]
  MoveL 613 to (58.44, 246.7, 260) mm, rotated rx -90 ry -25 rz 127.18 deg; joints [-3.358, -48.877, 103.874, -142.911, 108.539, -181.995, -1247.181]
  MoveL 614 to (58.8, 250.28, 270) mm, rotated rx -90 ry -25 rz 130.62 deg; joints [-2.992, -48.722, 103.605, -142.691, 108.575, -182.244, -1250.615]
  MoveL 615 to (58.94, 253.36, 280) mm, rotated rx -90 ry -25 rz 133.57 deg; joints [-2.628, -48.567, 103.33, -142.474, 108.608, -182.497, -1253.568]
  MoveL 616 to (58.93, 255.88, 290) mm, rotated rx -90 ry -25 rz 136 deg; joints [-2.265, -48.411, 103.049, -142.26, 108.636, -182.753, -1255.998]
  Set speed (1000.0 mm/s)
  MoveL 617 to (58.93, 255.88, 290) mm, rotated rx -90 ry -25 rz 136 deg; joints [-2.265, -48.411, 103.049, -142.26, 108.636, -182.753, -1255.998]
  Set speed (1000.0 mm/s)
  MoveL 618 to (37.11, 300.24, 290) mm, rotated rx -96.9 ry -17.88 rz 75.79 deg; joints [-6.114, -30.075, 34.443, -39.411, 47.865, -327.788, -1286.629]
  MoveL 619 to (37.11, 300.24, 290) mm, rotated rx -96.9 ry -17.88 rz 75.79 deg; joints [-6.114, -30.075, 34.443, -39.411, 47.865, -327.788, -1286.629]
  Set speed (60.0 mm/s)
  MoveL 620 to (39.03, 298.61, 280) mm, rotated rx -98.71 ry -16.79 rz 70.34 deg; joints [-6.407, -27.148, 28.965, -34.934, 50.939, -334.592, -1283.609]
  MoveL 621 to (41.29, 296.51, 270) mm, rotated rx -100.57 ry -16.08 rz 63.8 deg; joints [-6.657, -21.262, 17.719, -30.135, 57.401, -342.606, -1280.035]
  MoveL 622 to (43.78, 293.91, 260) mm, rotated rx -100.6 ry -13.96 rz 65.48 deg; joints [-6.933, -32.413, 38.828, -36.061, 43.052, -333.355, -1275.959]
  MoveL 623 to (46.4, 290.79, 250) mm, rotated rx -102.48 ry -13.76 rz 57.03 deg; joints [-7.152, -27.649, 30.021, -30.595, 49.358, -341.709, -1271.425]
  MoveL 624 to (49.06, 287.12, 240) mm, rotated rx -75.01 ry -14.65 rz 147.83 deg; joints [-9.131, -49.28, 110.781, -156.675, 113.803, -164.225, -1266.478]
  MoveL 625 to (51.62, 282.9, 230) mm, rotated rx -75.3 ry -12.71 rz 137.52 deg; joints [-9.892, -51.841, 111.409, -159.504, 107.009, -166.807, -1261.161]
  MoveL 626 to (53.98, 278.14, 220) mm, rotated rx -73.63 ry -13.16 rz 135.62 deg; joints [-10.569, -50.052, 111.477, -159.308, 112.284, -163.126, -1255.515]
